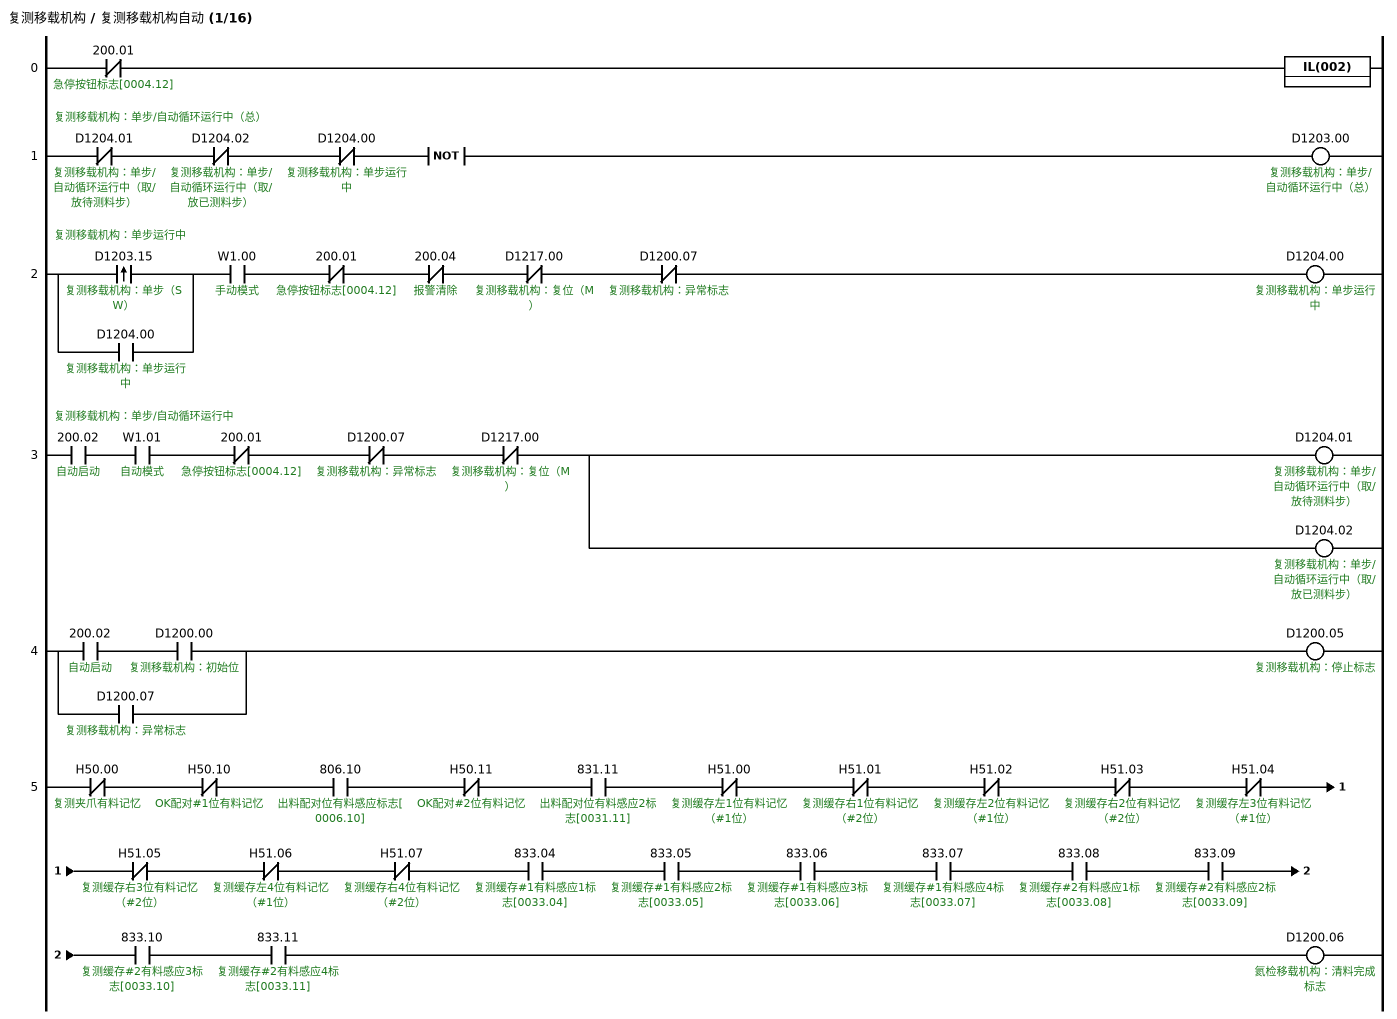
; [picture p528: 复测移载机构 / 复测移载机构自动, rungs 0-5]
; rung 0
LDNOT 200.01  ; 急停按钮标志[0004.12]
IL(002)
; rung 1: 复测移载机构：单步/自动循环运行中（总）
LDNOT D1204.01  ; 复测移载机构：单步/自动循环运行中（取/放待测料步）
ANDNOT D1204.02  ; 复测移载机构：单步/自动循环运行中（取/放已测料步）
ANDNOT D1204.00  ; 复测移载机构：单步运行中
NOT(520)
OUT D1203.00  ; 复测移载机构：单步/自动循环运行中（总）
; rung 2: 复测移载机构：单步运行中
@LD D1203.15  ; 复测移载机构：单步（SW）
OR D1204.00  ; 复测移载机构：单步运行中
AND W1.00  ; 手动模式
ANDNOT 200.01  ; 急停按钮标志[0004.12]
ANDNOT 200.04  ; 报警清除
ANDNOT D1217.00  ; 复测移载机构：复位（M）
ANDNOT D1200.07  ; 复测移载机构：异常标志
OUT D1204.00  ; 复测移载机构：单步运行中
; rung 3: 复测移载机构：单步/自动循环运行中
LD 200.02  ; 自动启动
AND W1.01  ; 自动模式
ANDNOT 200.01  ; 急停按钮标志[0004.12]
ANDNOT D1200.07  ; 复测移载机构：异常标志
ANDNOT D1217.00  ; 复测移载机构：复位（M）
OUT D1204.01  ; 复测移载机构：单步/自动循环运行中（取/放待测料步）
OUT D1204.02  ; 复测移载机构：单步/自动循环运行中（取/放已测料步）
; rung 4
LD 200.02  ; 自动启动
AND D1200.00  ; 复测移载机构：初始位
OR D1200.07  ; 复测移载机构：异常标志
OUT D1200.05  ; 复测移载机构：停止标志
; rung 5
LDNOT H50.00  ; 复测夹爪有料记忆
ANDNOT H50.10  ; OK配对#1位有料记忆
AND 806.10  ; 出料配对位有料感应标志[0006.10]
ANDNOT H50.11  ; OK配对#2位有料记忆
AND 831.11  ; 出料配对位有料感应2标志[0031.11]
ANDNOT H51.00  ; 复测缓存左1位有料记忆（#1位）
ANDNOT H51.01  ; 复测缓存右1位有料记忆（#2位）
ANDNOT H51.02  ; 复测缓存左2位有料记忆（#1位）
ANDNOT H51.03  ; 复测缓存右2位有料记忆（#2位）
ANDNOT H51.04  ; 复测缓存左3位有料记忆（#1位）
ANDNOT H51.05  ; 复测缓存右3位有料记忆（#2位）
ANDNOT H51.06  ; 复测缓存左4位有料记忆（#1位）
ANDNOT H51.07  ; 复测缓存右4位有料记忆（#2位）
AND 833.04  ; 复测缓存#1有料感应1标志[0033.04]
AND 833.05  ; 复测缓存#1有料感应2标志[0033.05]
AND 833.06  ; 复测缓存#1有料感应3标志[0033.06]
AND 833.07  ; 复测缓存#1有料感应4标志[0033.07]
AND 833.08  ; 复测缓存#2有料感应1标志[0033.08]
AND 833.09  ; 复测缓存#2有料感应2标志[0033.09]
AND 833.10  ; 复测缓存#2有料感应3标志[0033.10]
AND 833.11  ; 复测缓存#2有料感应4标志[0033.11]
OUT D1200.06  ; 氦检移载机构：清料完成标志

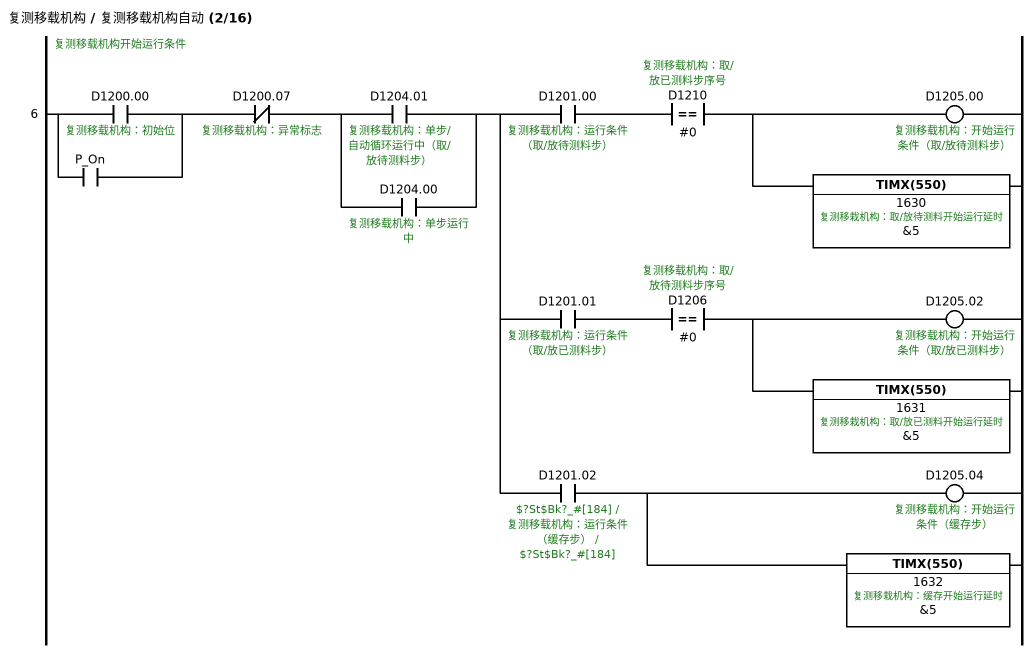
; rung 6: 复测移载机构开始运行条件
LD D1200.00  ; 复测移载机构：初始位
OR P_On
ANDNOT D1200.07  ; 复测移载机构：异常标志
LD D1204.01  ; 复测移载机构：单步/自动循环运行中（取/放待测料步）
OR D1204.00  ; 复测移载机构：单步运行中
ANDLD
OUT TR0
AND D1201.00  ; 复测移载机构：运行条件（取/放待测料步）
AND=L(301) D1210 #0  ; 复测移载机构：取/放已测料步序号
OUT D1205.00  ; 复测移载机构：开始运行条件（取/放待测料步）
TIMX(550) 1630 &5  ; 复测移栽机构：取/放待测料开始运行延时
LD TR0
AND D1201.01  ; 复测移载机构：运行条件（取/放已测料步）
AND=L(301) D1206 #0  ; 复测移载机构：取/放待测料步序号
OUT D1205.02  ; 复测移载机构：开始运行条件（取/放已测料步）
TIMX(550) 1631 &5  ; 复测移栽机构：取/放已测料开始运行延时
LD TR0
AND D1201.02  ; $?St$Bk?_#[184] / 复测移载机构：运行条件（缓存步） / $?St$Bk?_#[184]
OUT D1205.04  ; 复测移载机构：开始运行条件（缓存步）
TIMX(550) 1632 &5  ; 复测移栽机构：缓存开始运行延时

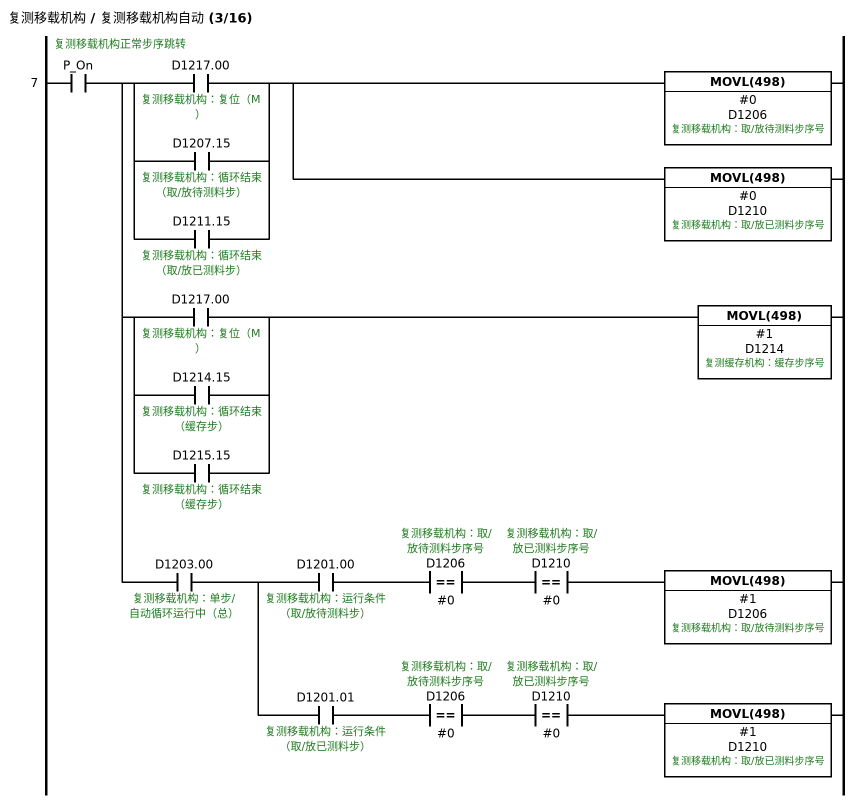
; rung 7: 复测移载机构正常步序跳转
LD P_On
OUT TR0
LD D1217.00  ; 复测移载机构：复位（M）
OR D1207.15  ; 复测移载机构：循环结束（取/放待测料步）
OR D1211.15  ; 复测移载机构：循环结束（取/放已测料步）
ANDLD
MOVL(498) #0 D1206  ; 复测移载机构：取/放待测料步序号
MOVL(498) #0 D1210  ; 复测移载机构：取/放已测料步序号
LD TR0
LD D1217.00  ; 复测移载机构：复位（M）
OR D1214.15  ; 复测移载机构：循环结束（缓存步）
OR D1215.15  ; 复测移载机构：循环结束（缓存步）
ANDLD
MOVL(498) #1 D1214  ; 复测缓存机构：缓存步序号
LD TR0
AND D1203.00  ; 复测移载机构：单步/自动循环运行中（总）
OUT TR0
AND D1201.00  ; 复测移载机构：运行条件（取/放待测料步）
AND=L(301) D1206 #0  ; 复测移载机构：取/放待测料步序号
AND=L(301) D1210 #0  ; 复测移载机构：取/放已测料步序号
MOVL(498) #1 D1206  ; 复测移载机构：取/放待测料步序号
LD TR0
AND D1201.01  ; 复测移载机构：运行条件（取/放已测料步）
AND=L(301) D1206 #0  ; 复测移载机构：取/放待测料步序号
AND=L(301) D1210 #0  ; 复测移载机构：取/放已测料步序号
MOVL(498) #1 D1210  ; 复测移载机构：取/放已测料步序号

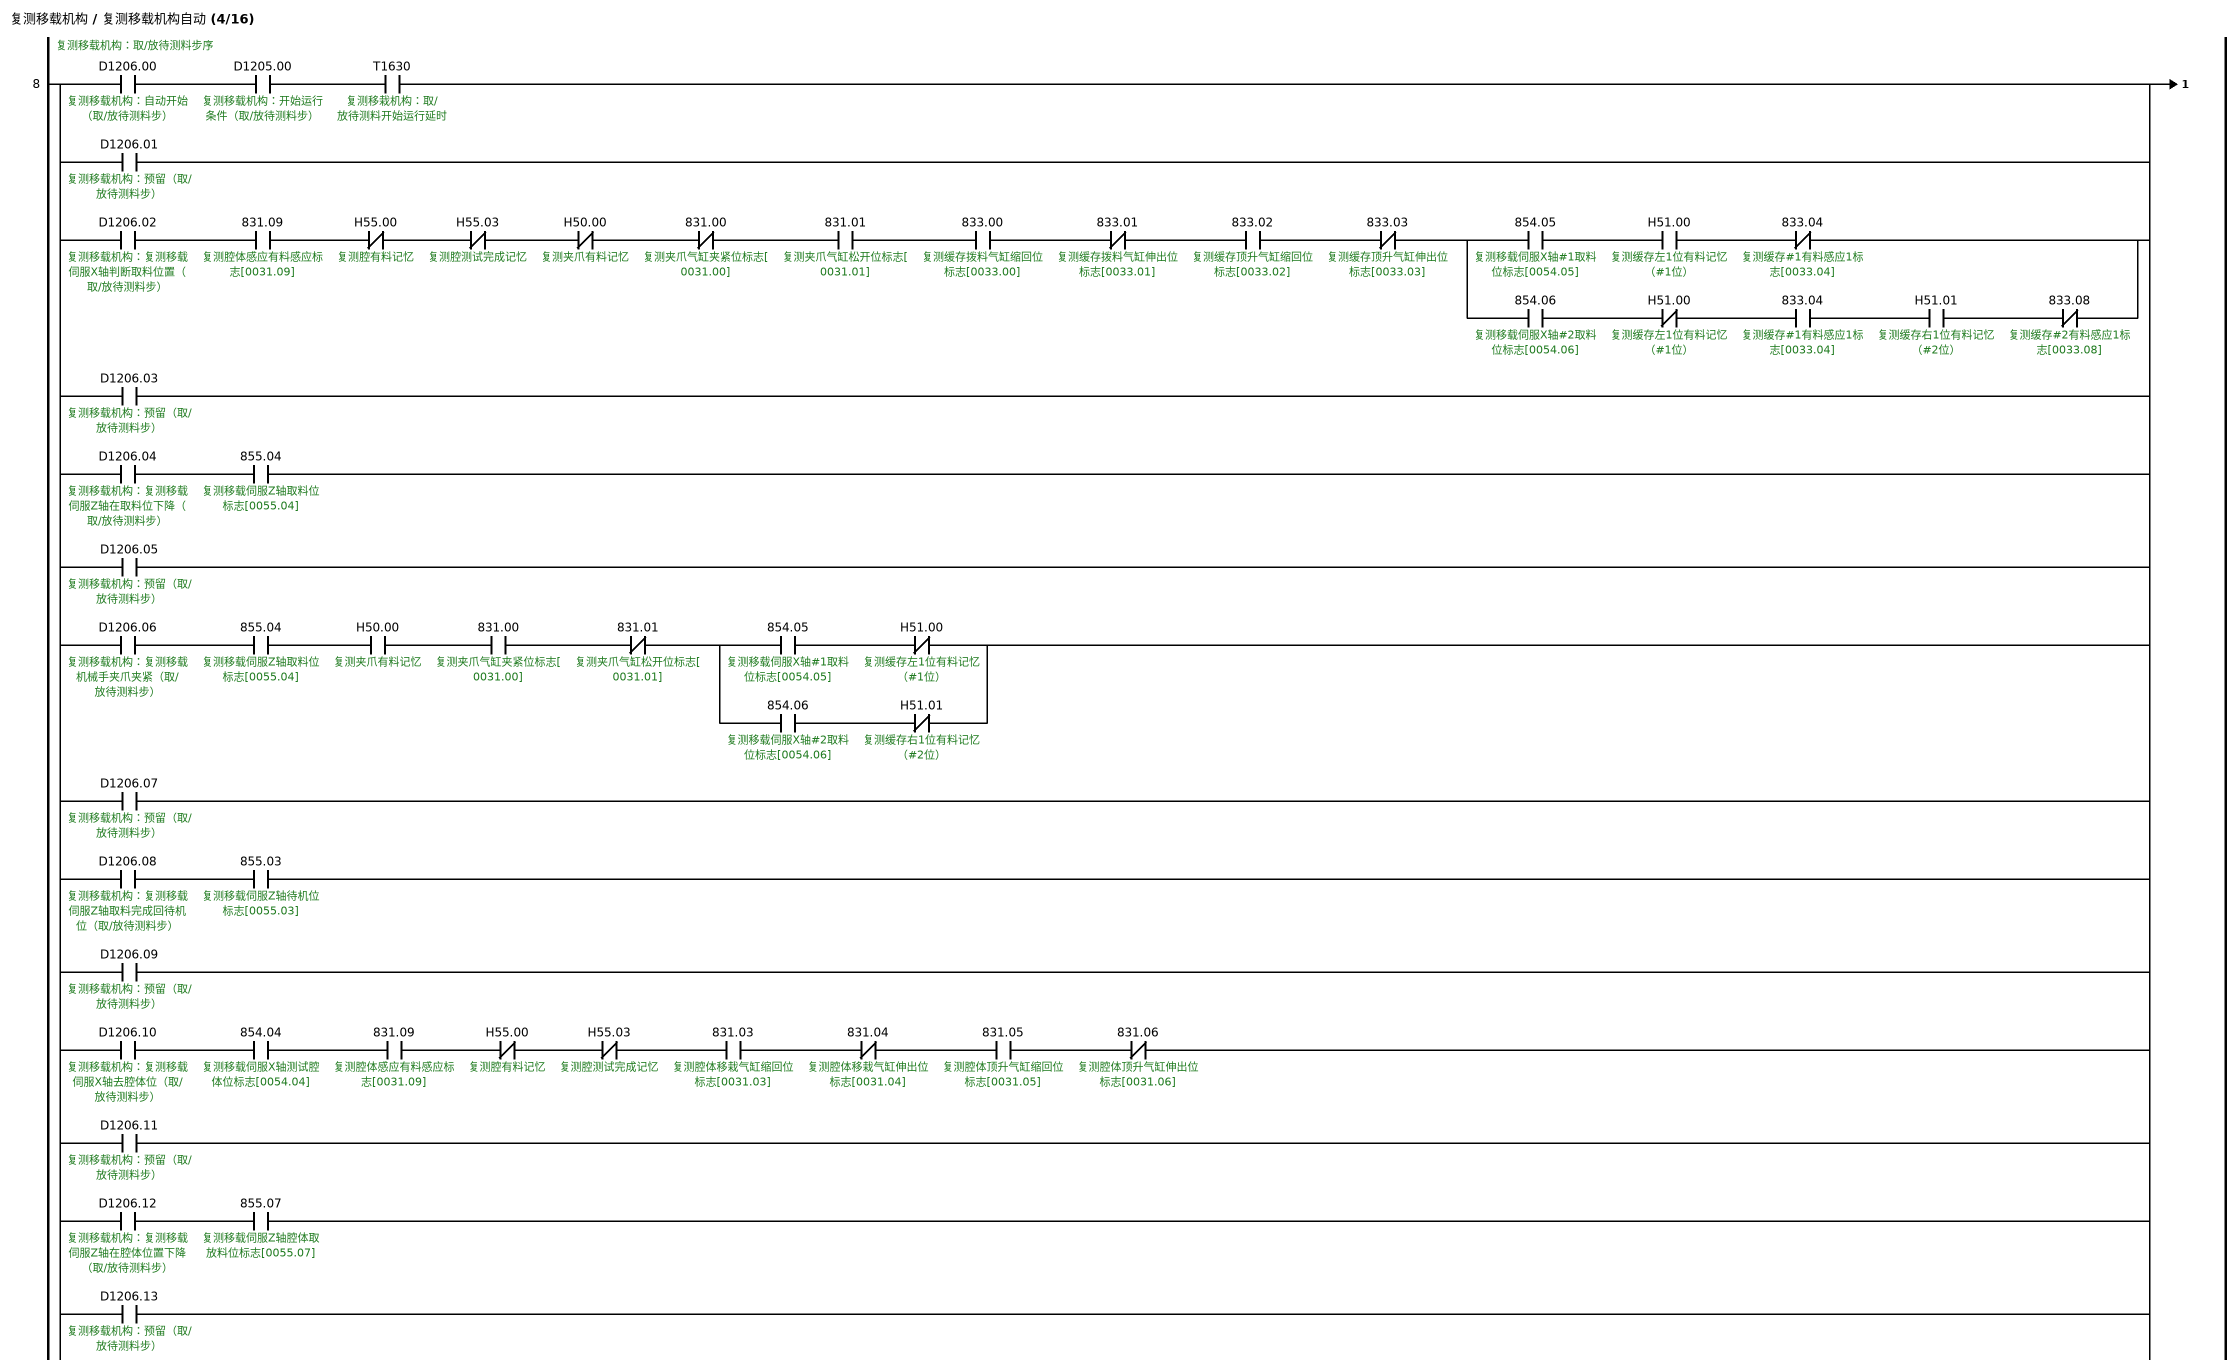

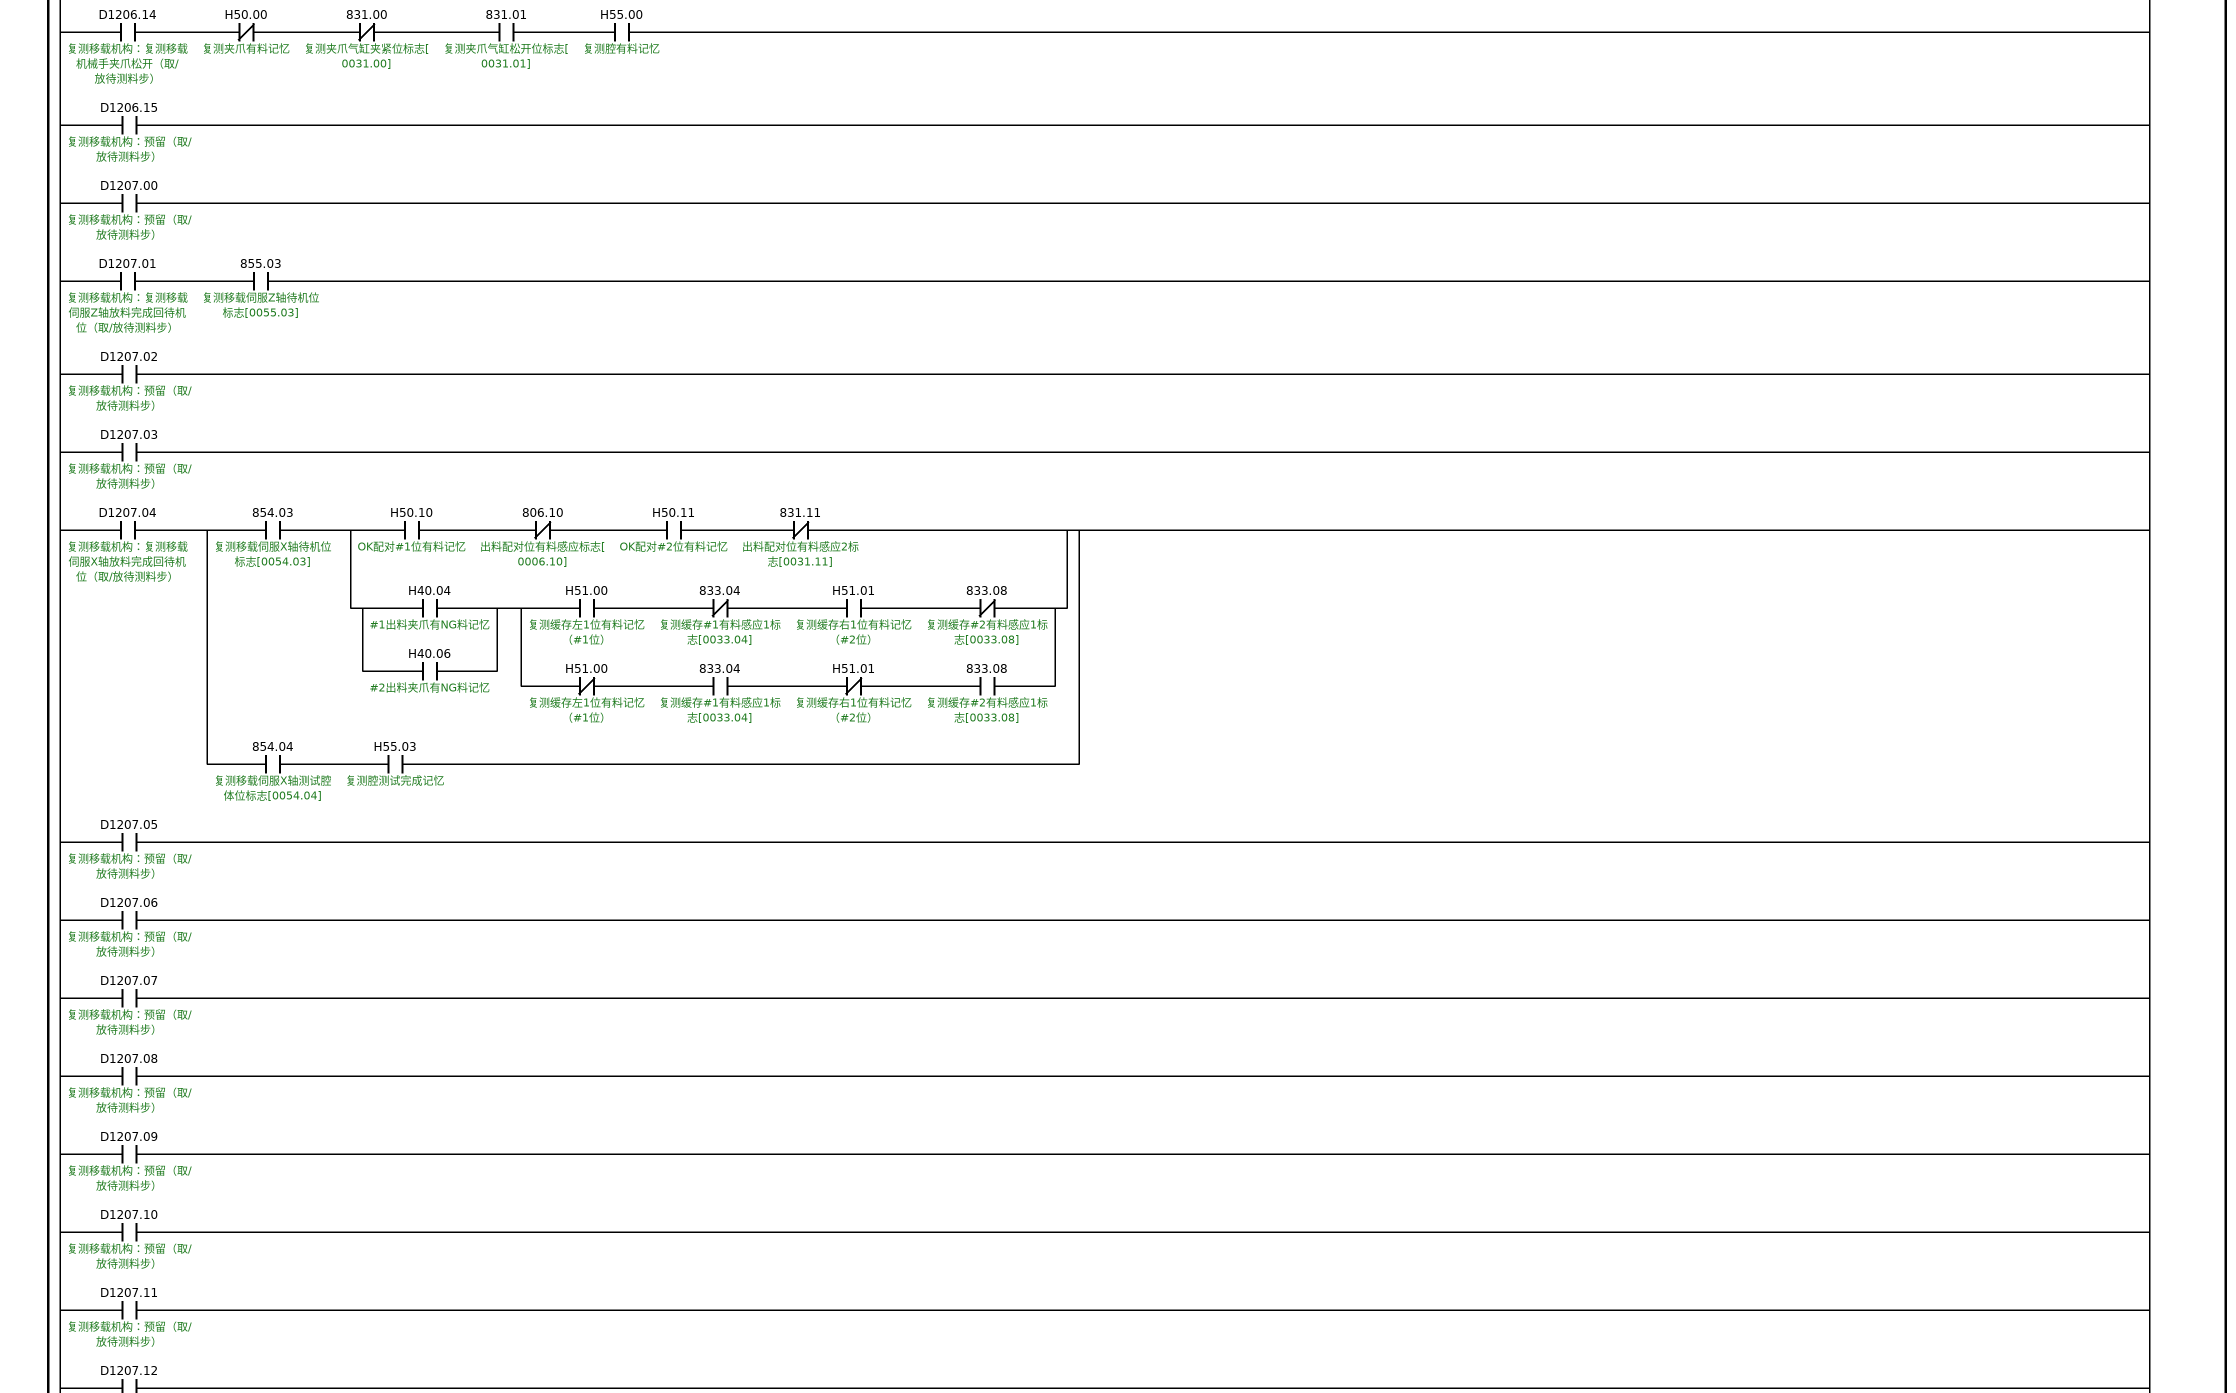

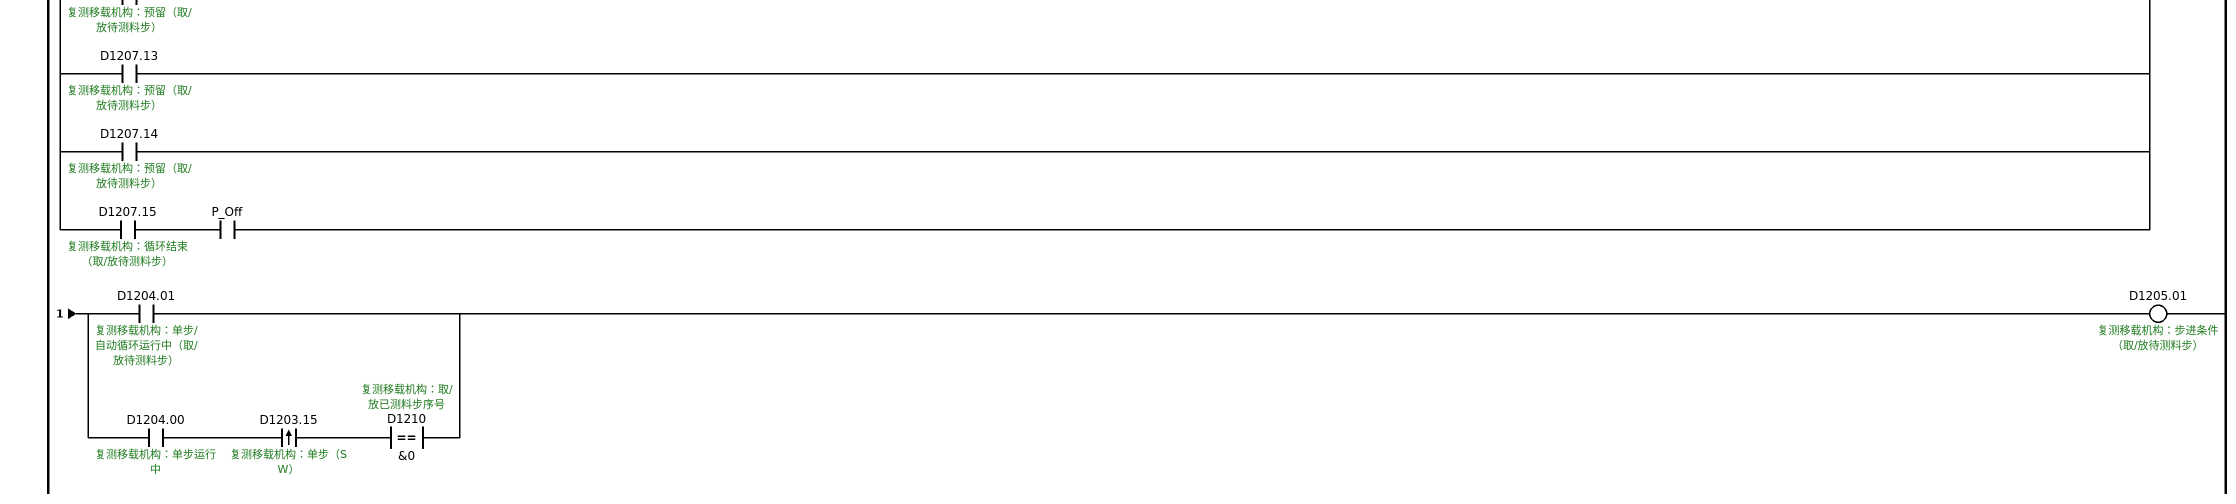
; rung 8: 复测移载机构：取/放待测料步序
LD D1206.00  ; 复测移载机构：自动开始（取/放待测料步）
AND D1205.00  ; 复测移载机构：开始运行条件（取/放待测料步）
AND T1630  ; 复测移栽机构：取/放待测料开始运行延时
OR D1206.01  ; 复测移载机构：预留（取/放待测料步）
LD D1206.02  ; 复测移载机构：复测移载伺服X轴判断取料位置（取/放待测料步）  // 如果出现带料初始化时，夹爪有料，则直接跳转至腔体放料步（D1206.10）
AND 831.09  ; 复测腔体感应有料感应标志[0031.09]
ANDNOT H55.00  ; 复测腔有料记忆
ANDNOT H55.03  ; 复测腔测试完成记忆
ANDNOT H50.00  ; 复测夹爪有料记忆
ANDNOT 831.00  ; 复测夹爪气缸夹紧位标志[0031.00]
AND 831.01  ; 复测夹爪气缸松开位标志[0031.01]
AND 833.00  ; 复测缓存拨料气缸缩回位标志[0033.00]
ANDNOT 833.01  ; 复测缓存拨料气缸伸出位标志[0033.01]
AND 833.02  ; 复测缓存顶升气缸缩回位标志[0033.02]
ANDNOT 833.03  ; 复测缓存顶升气缸伸出位标志[0033.03]
LD 854.05  ; 复测移载伺服X轴#1取料位标志[0054.05]
AND H51.00  ; 复测缓存左1位有料记忆（#1位）
ANDNOT 833.04  ; 复测缓存#1有料感应1标志[0033.04]
LD 854.06  ; 复测移载伺服X轴#2取料位标志[0054.06]
ANDNOT H51.00  ; 复测缓存左1位有料记忆（#1位）
AND 833.04  ; 复测缓存#1有料感应1标志[0033.04]
AND H51.01  ; 复测缓存右1位有料记忆（#2位）
ANDNOT 833.08  ; 复测缓存#2有料感应1标志[0033.08]
ORLD
ANDLD
ORLD
OR D1206.03  ; 复测移载机构：预留（取/放待测料步）
LD D1206.04  ; 复测移载机构：复测移载伺服Z轴在取料位下降（取/放待测料步）
AND 855.04  ; 复测移载伺服Z轴取料位标志[0055.04]
ORLD
OR D1206.05  ; 复测移载机构：预留（取/放待测料步）
LD D1206.06  ; 复测移载机构：复测移载机械手夹爪夹紧（取/放待测料步）
AND 855.04  ; 复测移载伺服Z轴取料位标志[0055.04]
AND H50.00  ; 复测夹爪有料记忆
AND 831.00  ; 复测夹爪气缸夹紧位标志[0031.00]
ANDNOT 831.01  ; 复测夹爪气缸松开位标志[0031.01]
LD 854.05  ; 复测移载伺服X轴#1取料位标志[0054.05]
ANDNOT H51.00  ; 复测缓存左1位有料记忆（#1位）
LD 854.06  ; 复测移载伺服X轴#2取料位标志[0054.06]
ANDNOT H51.01  ; 复测缓存右1位有料记忆（#2位）
ORLD
ANDLD
ORLD
OR D1206.07  ; 复测移载机构：预留（取/放待测料步）
LD D1206.08  ; 复测移载机构：复测移载伺服Z轴取料完成回待机位（取/放待测料步）
AND 855.03  ; 复测移载伺服Z轴待机位标志[0055.03]
ORLD
OR D1206.09  ; 复测移载机构：预留（取/放待测料步）
LD D1206.10  ; 复测移载机构：复测移载伺服X轴去腔体位（取/放待测料步）
AND 854.04  ; 复测移载伺服X轴测试腔体位标志[0054.04]
AND 831.09  ; 复测腔体感应有料感应标志[0031.09]
ANDNOT H55.00  ; 复测腔有料记忆
ANDNOT H55.03  ; 复测腔测试完成记忆
AND 831.03  ; 复测腔体移栽气缸缩回位标志[0031.03]
ANDNOT 831.04  ; 复测腔体移栽气缸伸出位标志[0031.04]
AND 831.05  ; 复测腔体顶升气缸缩回位标志[0031.05]
ANDNOT 831.06  ; 复测腔体顶升气缸伸出位标志[0031.06]
ORLD
OR D1206.11  ; 复测移载机构：预留（取/放待测料步）
LD D1206.12  ; 复测移载机构：复测移载伺服Z轴在腔体位置下降（取/放待测料步）
AND 855.07  ; 复测移载伺服Z轴腔体取放料位标志[0055.07]
ORLD
OR D1206.13  ; 复测移载机构：预留（取/放待测料步）
LD D1206.14  ; 复测移载机构：复测移载机械手夹爪松开（取/放待测料步）
ANDNOT H50.00  ; 复测夹爪有料记忆
ANDNOT 831.00  ; 复测夹爪气缸夹紧位标志[0031.00]
AND 831.01  ; 复测夹爪气缸松开位标志[0031.01]
AND H55.00  ; 复测腔有料记忆
ORLD
OR D1206.15  ; 复测移载机构：预留（取/放待测料步）
OR D1207.00  ; 复测移载机构：预留（取/放待测料步）
LD D1207.01  ; 复测移载机构：复测移载伺服Z轴放料完成回待机位（取/放待测料步）
AND 855.03  ; 复测移载伺服Z轴待机位标志[0055.03]
ORLD
OR D1207.02  ; 复测移载机构：预留（取/放待测料步）
OR D1207.03  ; 复测移载机构：预留（取/放待测料步）
LD D1207.04  ; 复测移载机构：复测移载伺服X轴放料完成回待机位（取/放待测料步）  // 当配对位有空位，且缓存位有单料时在腔体位等待
LD 854.03  ; 复测移载伺服X轴待机位标志[0054.03]
LD H50.10  ; OK配对#1位有料记忆
ANDNOT 806.10  ; 出料配对位有料感应标志[0006.10]
AND H50.11  ; OK配对#2位有料记忆
ANDNOT 831.11  ; 出料配对位有料感应2标志[0031.11]
LD H40.04  ; #1出料夹爪有NG料记忆
OR H40.06  ; #2出料夹爪有NG料记忆
LD H51.00  ; 复测缓存左1位有料记忆（#1位）
ANDNOT 833.04  ; 复测缓存#1有料感应1标志[0033.04]
AND H51.01  ; 复测缓存右1位有料记忆（#2位）
ANDNOT 833.08  ; 复测缓存#2有料感应1标志[0033.08]
LDNOT H51.00  ; 复测缓存左1位有料记忆（#1位）
AND 833.04  ; 复测缓存#1有料感应1标志[0033.04]
ANDNOT H51.01  ; 复测缓存右1位有料记忆（#2位）
AND 833.08  ; 复测缓存#2有料感应1标志[0033.08]
ORLD
ANDLD
ORLD
ANDLD
LD 854.04  ; 复测移载伺服X轴测试腔体位标志[0054.04]
AND H55.03  ; 复测腔测试完成记忆
ORLD
ANDLD
ORLD
OR D1207.05  ; 复测移载机构：预留（取/放待测料步）
OR D1207.06  ; 复测移载机构：预留（取/放待测料步）
OR D1207.07  ; 复测移载机构：预留（取/放待测料步）
OR D1207.08  ; 复测移载机构：预留（取/放待测料步）
OR D1207.09  ; 复测移载机构：预留（取/放待测料步）
OR D1207.10  ; 复测移载机构：预留（取/放待测料步）
OR D1207.11  ; 复测移载机构：预留（取/放待测料步）
OR D1207.12  ; 复测移载机构：预留（取/放待测料步）
OR D1207.13  ; 复测移载机构：预留（取/放待测料步）
OR D1207.14  ; 复测移载机构：预留（取/放待测料步）
LD D1207.15  ; 复测移载机构：循环结束（取/放待测料步）
AND P_Off
ORLD
LD D1204.01  ; 复测移载机构：单步/自动循环运行中（取/放待测料步）
LD D1204.00  ; 复测移载机构：单步运行中
@AND D1203.15  ; 复测移载机构：单步（SW）
AND=L(301) D1210 &0  ; 复测移载机构：取/放已测料步序号
ORLD
ANDLD
OUT D1205.01  ; 复测移载机构：步进条件（取/放待测料步）

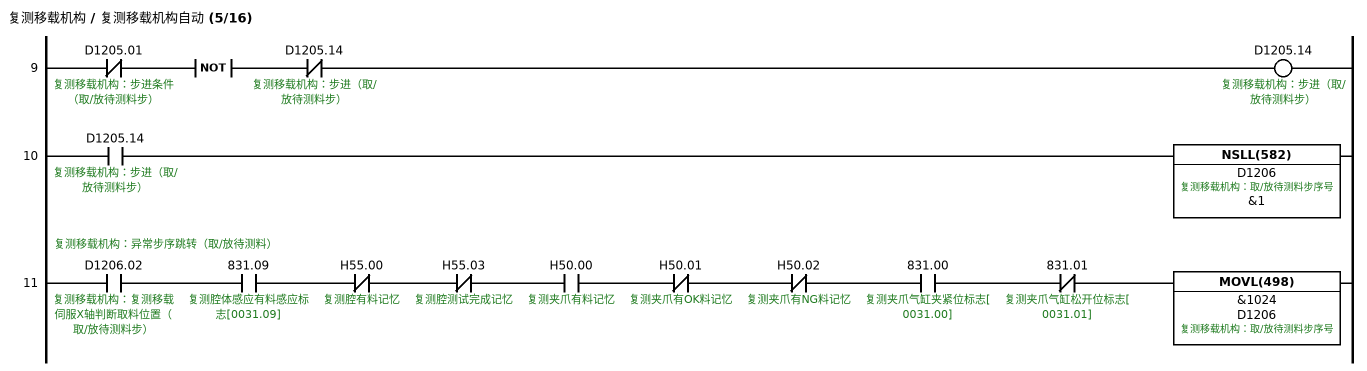
; rung 9
LDNOT D1205.01  ; 复测移载机构：步进条件（取/放待测料步）
NOT(520)
ANDNOT D1205.14  ; 复测移载机构：步进（取/放待测料步）
OUT D1205.14  ; 复测移载机构：步进（取/放待测料步）
; rung 10
LD D1205.14  ; 复测移载机构：步进（取/放待测料步）
NSLL(582) D1206 &1  ; 复测移载机构：取/放待测料步序号
; rung 11: 复测移载机构：异常步序跳转（取/放待测料）
LD D1206.02  ; 复测移载机构：复测移载伺服X轴判断取料位置（取/放待测料步）  // 如果出现带料初始化时，夹爪有料，则直接跳转至腔体放料步（D1206.10）
AND 831.09  ; 复测腔体感应有料感应标志[0031.09]
ANDNOT H55.00  ; 复测腔有料记忆
ANDNOT H55.03  ; 复测腔测试完成记忆
AND H50.00  ; 复测夹爪有料记忆
ANDNOT H50.01  ; 复测夹爪有OK料记忆
ANDNOT H50.02  ; 复测夹爪有NG料记忆
AND 831.00  ; 复测夹爪气缸夹紧位标志[0031.00]
ANDNOT 831.01  ; 复测夹爪气缸松开位标志[0031.01]
MOVL(498) &1024 D1206  ; 复测移载机构：取/放待测料步序号

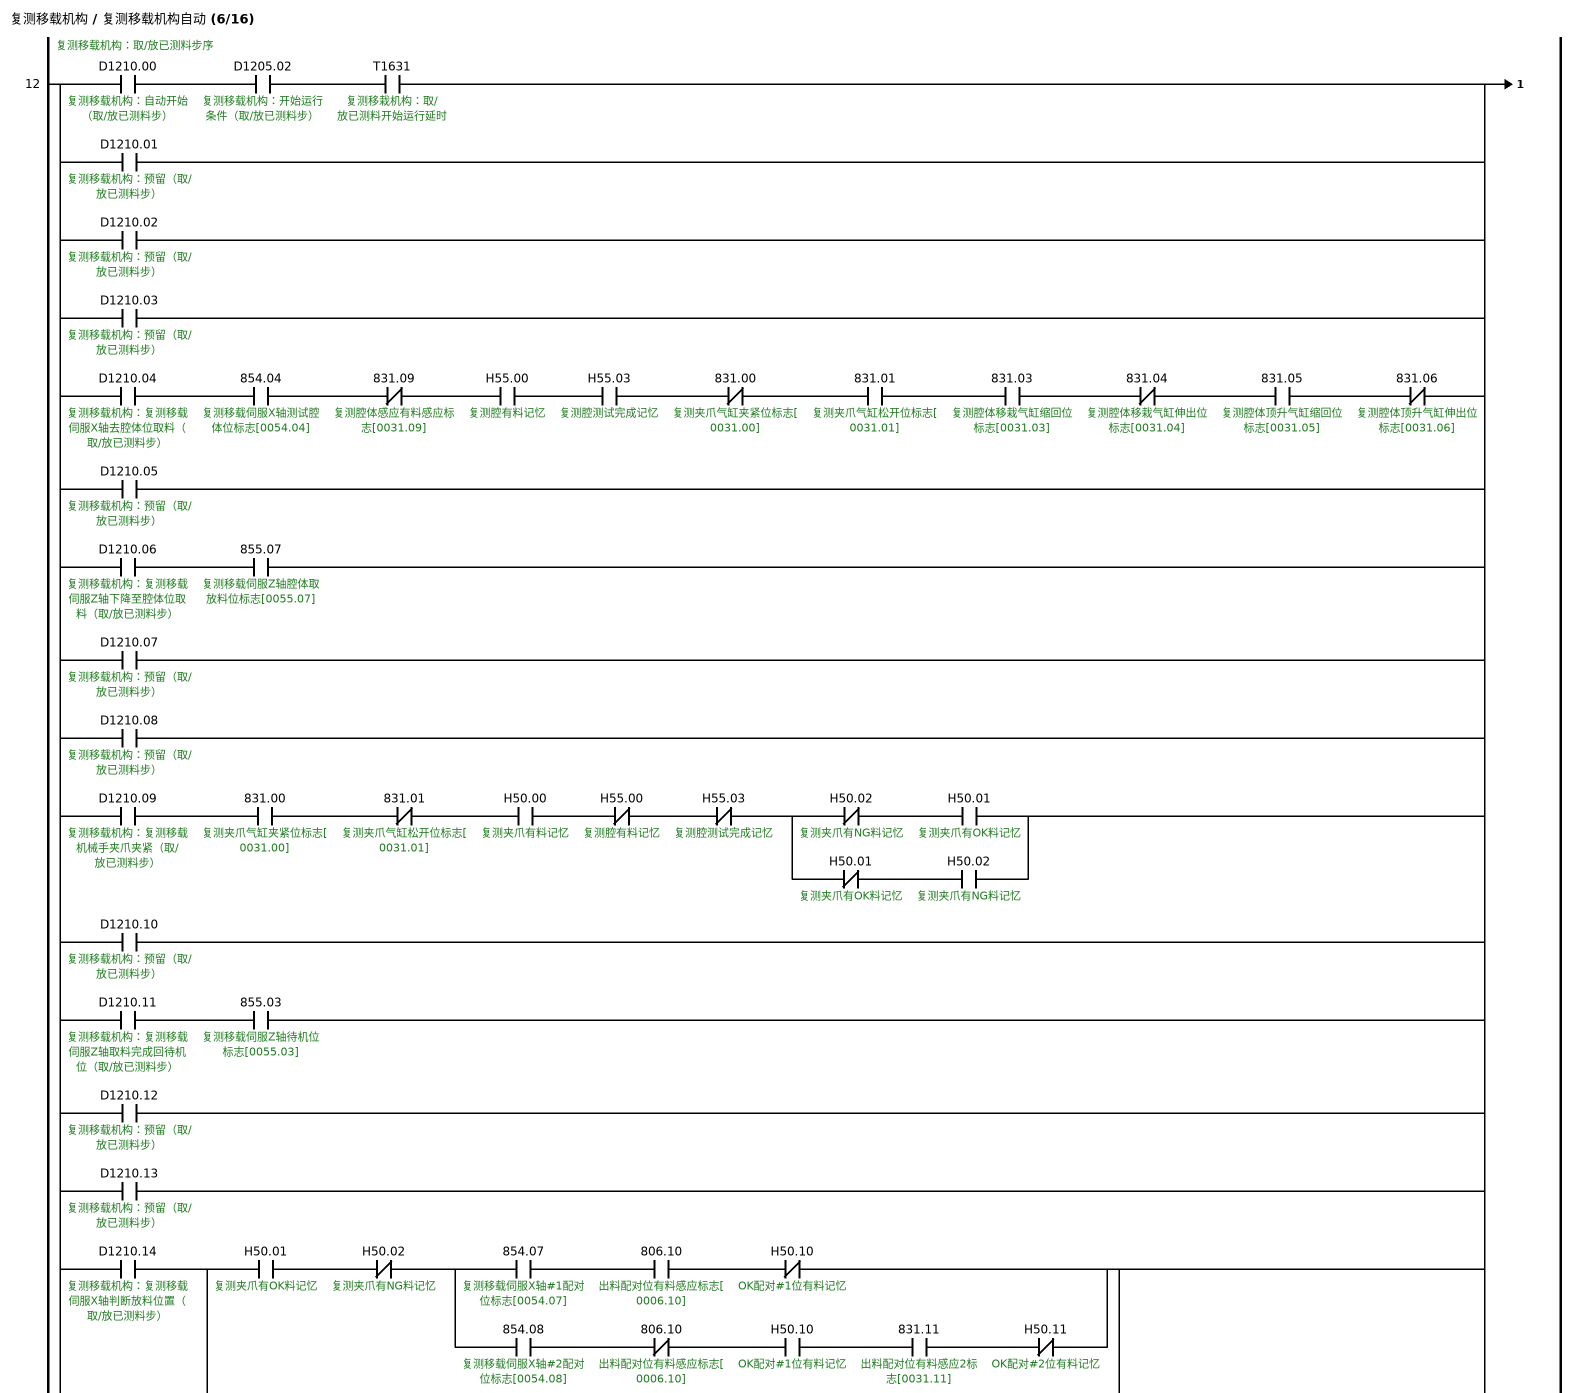

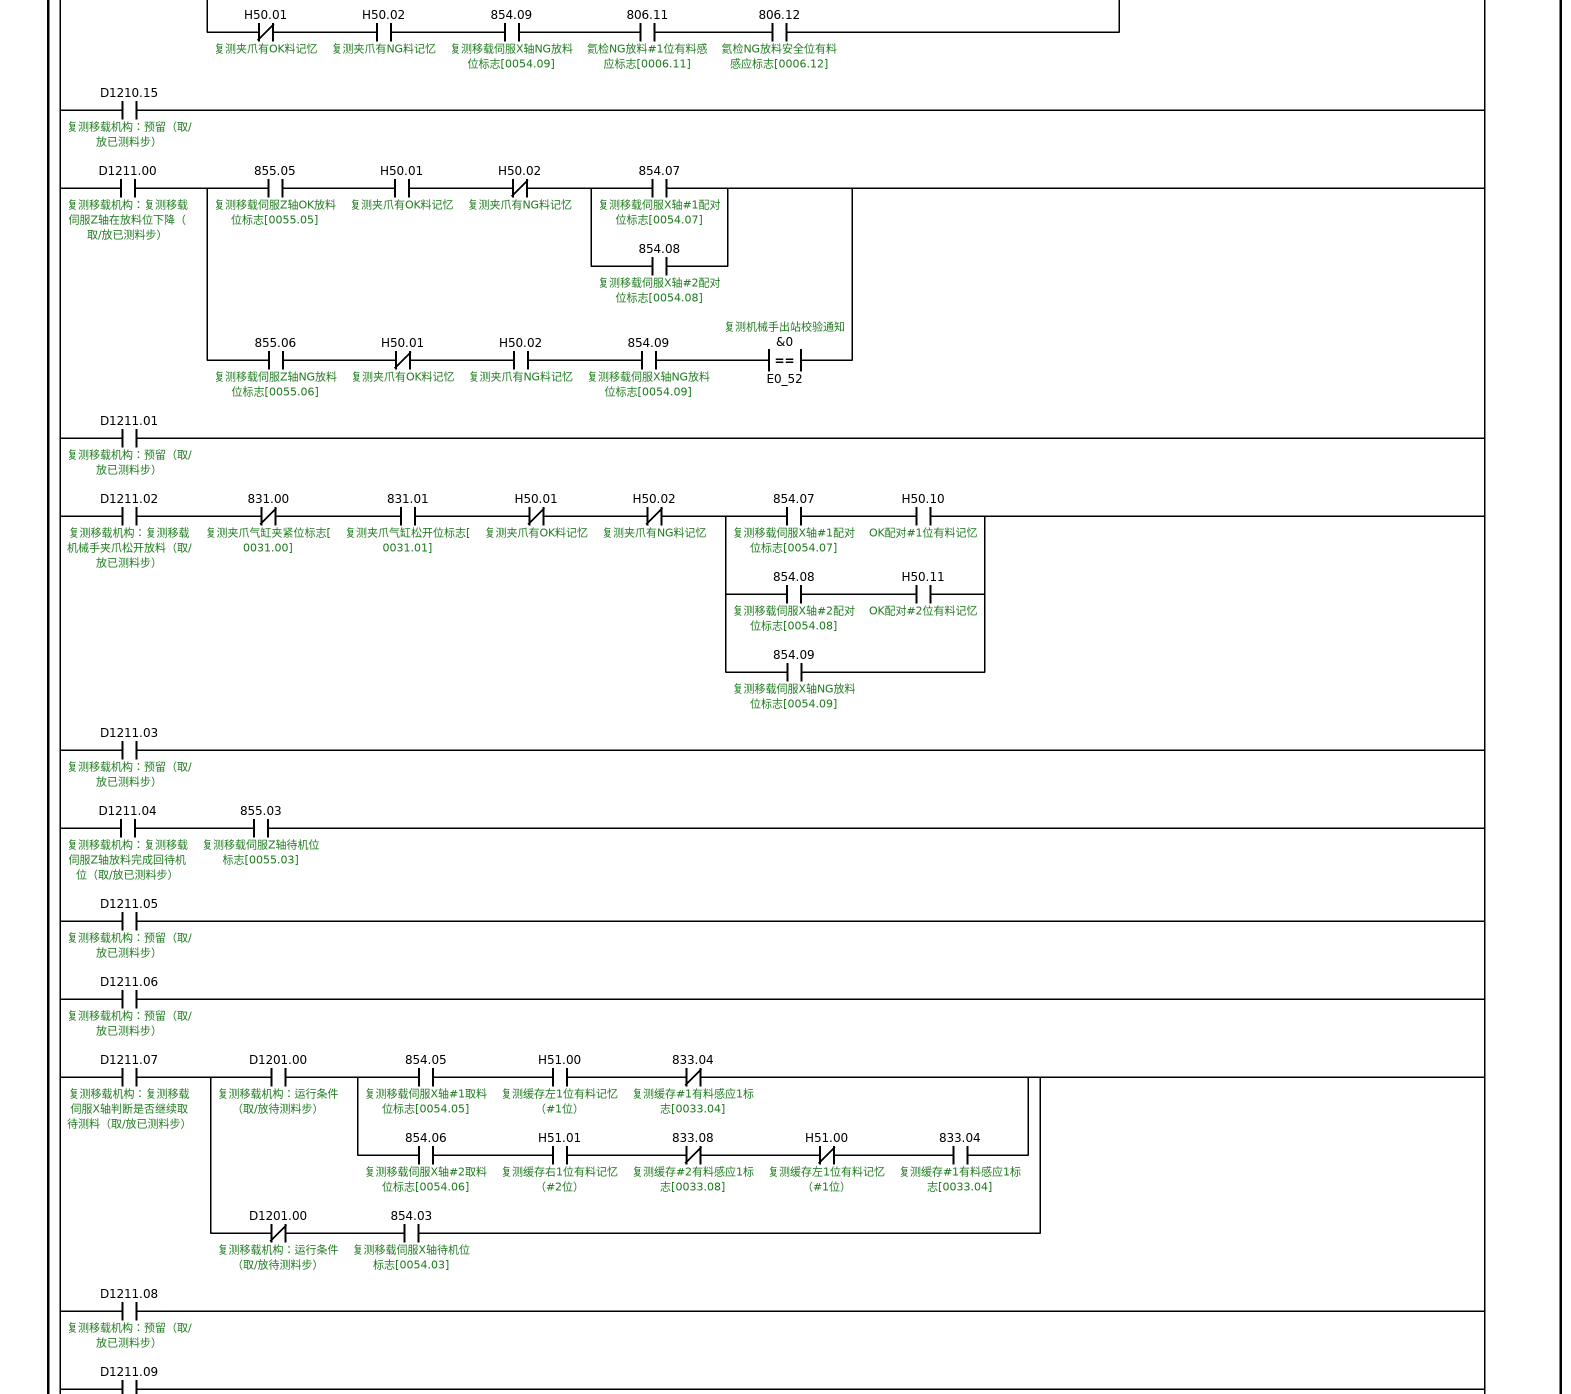

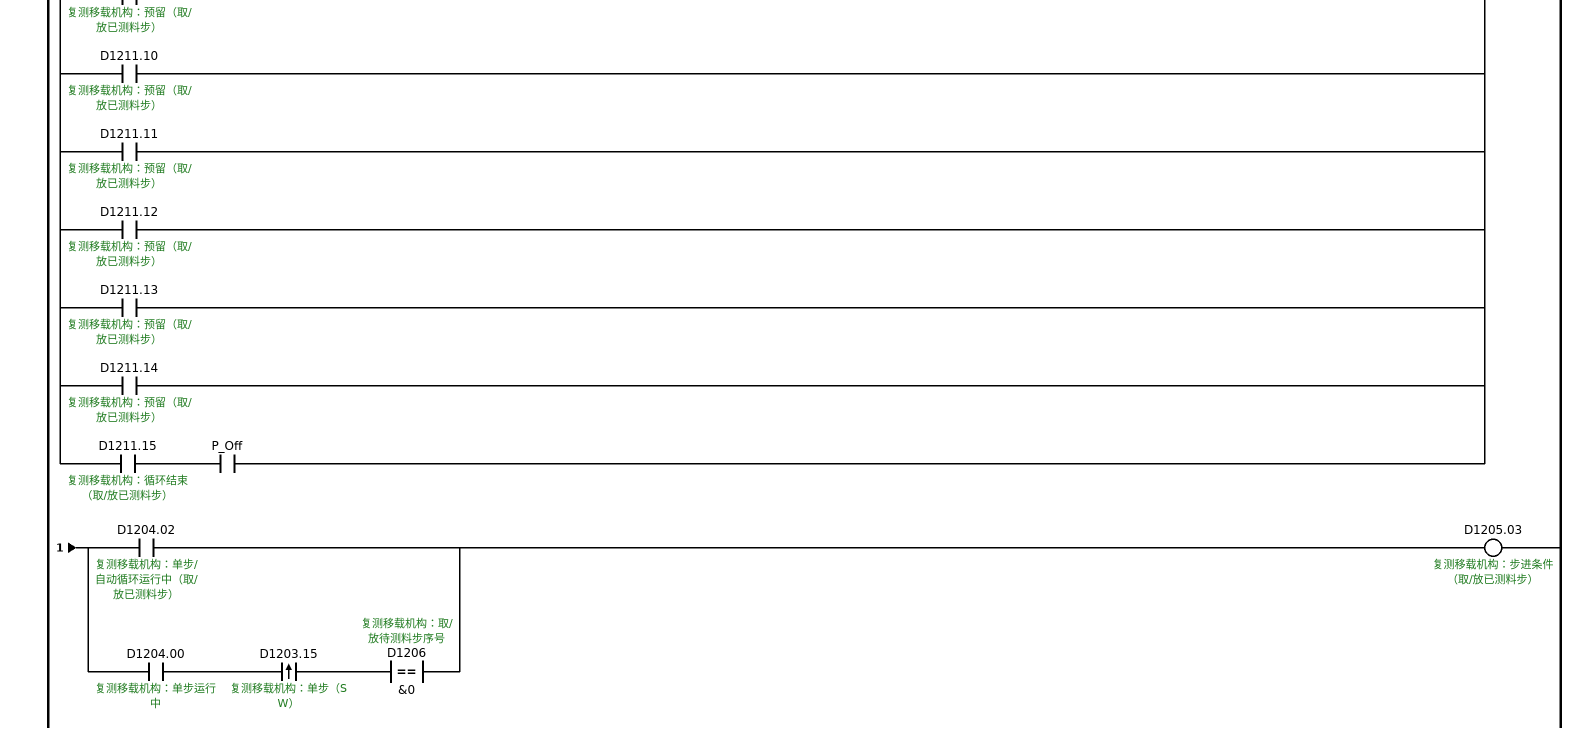
; rung 12: 复测移载机构：取/放已测料步序
LD D1210.00  ; 复测移载机构：自动开始（取/放已测料步）
AND D1205.02  ; 复测移载机构：开始运行条件（取/放已测料步）
AND T1631  ; 复测移栽机构：取/放已测料开始运行延时
OR D1210.01  ; 复测移载机构：预留（取/放已测料步）
OR D1210.02  ; 复测移载机构：预留（取/放已测料步）
OR D1210.03  ; 复测移载机构：预留（取/放已测料步）
LD D1210.04  ; 复测移载机构：复测移载伺服X轴去腔体位取料（取/放已测料步）  // 如果出现带料初始化时，夹爪有料，则直接跳转至放料判断步（D1210.14）
AND 854.04  ; 复测移载伺服X轴测试腔体位标志[0054.04]
ANDNOT 831.09  ; 复测腔体感应有料感应标志[0031.09]
AND H55.00  ; 复测腔有料记忆
AND H55.03  ; 复测腔测试完成记忆
ANDNOT 831.00  ; 复测夹爪气缸夹紧位标志[0031.00]
AND 831.01  ; 复测夹爪气缸松开位标志[0031.01]
AND 831.03  ; 复测腔体移栽气缸缩回位标志[0031.03]
ANDNOT 831.04  ; 复测腔体移栽气缸伸出位标志[0031.04]
AND 831.05  ; 复测腔体顶升气缸缩回位标志[0031.05]
ANDNOT 831.06  ; 复测腔体顶升气缸伸出位标志[0031.06]
ORLD
OR D1210.05  ; 复测移载机构：预留（取/放已测料步）
LD D1210.06  ; 复测移载机构：复测移载伺服Z轴下降至腔体位取料（取/放已测料步）
AND 855.07  ; 复测移载伺服Z轴腔体取放料位标志[0055.07]
ORLD
OR D1210.07  ; 复测移载机构：预留（取/放已测料步）
OR D1210.08  ; 复测移载机构：预留（取/放已测料步）
LD D1210.09  ; 复测移载机构：复测移载机械手夹爪夹紧（取/放已测料步）
AND 831.00  ; 复测夹爪气缸夹紧位标志[0031.00]
ANDNOT 831.01  ; 复测夹爪气缸松开位标志[0031.01]
AND H50.00  ; 复测夹爪有料记忆
ANDNOT H55.00  ; 复测腔有料记忆
ANDNOT H55.03  ; 复测腔测试完成记忆
LDNOT H50.02  ; 复测夹爪有NG料记忆
AND H50.01  ; 复测夹爪有OK料记忆
LDNOT H50.01  ; 复测夹爪有OK料记忆
AND H50.02  ; 复测夹爪有NG料记忆
ORLD
ANDLD
ORLD
OR D1210.10  ; 复测移载机构：预留（取/放已测料步）
LD D1210.11  ; 复测移载机构：复测移载伺服Z轴取料完成回待机位（取/放已测料步）
AND 855.03  ; 复测移载伺服Z轴待机位标志[0055.03]
ORLD
OR D1210.12  ; 复测移载机构：预留（取/放已测料步）
OR D1210.13  ; 复测移载机构：预留（取/放已测料步）
LD D1210.14  ; 复测移载机构：复测移载伺服X轴判断放料位置（取/放已测料步）
LD H50.01  ; 复测夹爪有OK料记忆
ANDNOT H50.02  ; 复测夹爪有NG料记忆
LD 854.07  ; 复测移载伺服X轴#1配对位标志[0054.07]
AND 806.10  ; 出料配对位有料感应标志[0006.10]
ANDNOT H50.10  ; OK配对#1位有料记忆
LD 854.08  ; 复测移载伺服X轴#2配对位标志[0054.08]
ANDNOT 806.10  ; 出料配对位有料感应标志[0006.10]
AND H50.10  ; OK配对#1位有料记忆
AND 831.11  ; 出料配对位有料感应2标志[0031.11]
ANDNOT H50.11  ; OK配对#2位有料记忆
ORLD
ANDLD
LDNOT H50.01  ; 复测夹爪有OK料记忆
AND H50.02  ; 复测夹爪有NG料记忆
AND 854.09  ; 复测移载伺服X轴NG放料位标志[0054.09]
AND 806.11  ; 氦检NG放料#1位有料感应标志[0006.11]
AND 806.12  ; 氦检NG放料安全位有料感应标志[0006.12]
ORLD
ANDLD
ORLD
OR D1210.15  ; 复测移载机构：预留（取/放已测料步）
LD D1211.00  ; 复测移载机构：复测移载伺服Z轴在放料位下降（取/放已测料步）
LD 855.05  ; 复测移载伺服Z轴OK放料位标志[0055.05]
AND H50.01  ; 复测夹爪有OK料记忆
ANDNOT H50.02  ; 复测夹爪有NG料记忆
LD 854.07  ; 复测移载伺服X轴#1配对位标志[0054.07]
OR 854.08  ; 复测移载伺服X轴#2配对位标志[0054.08]
ANDLD
LD 855.06  ; 复测移载伺服Z轴NG放料位标志[0055.06]
ANDNOT H50.01  ; 复测夹爪有OK料记忆
AND H50.02  ; 复测夹爪有NG料记忆
AND 854.09  ; 复测移载伺服X轴NG放料位标志[0054.09]
AND=(300) &0 E0_52  ; 复测机械手出站校验通知
ORLD
ANDLD
ORLD
OR D1211.01  ; 复测移载机构：预留（取/放已测料步）
LD D1211.02  ; 复测移载机构：复测移载机械手夹爪松开放料（取/放已测料步）
ANDNOT 831.00  ; 复测夹爪气缸夹紧位标志[0031.00]
AND 831.01  ; 复测夹爪气缸松开位标志[0031.01]
ANDNOT H50.01  ; 复测夹爪有OK料记忆
ANDNOT H50.02  ; 复测夹爪有NG料记忆
LD 854.07  ; 复测移载伺服X轴#1配对位标志[0054.07]
AND H50.10  ; OK配对#1位有料记忆
LD 854.08  ; 复测移载伺服X轴#2配对位标志[0054.08]
AND H50.11  ; OK配对#2位有料记忆
ORLD
OR 854.09  ; 复测移载伺服X轴NG放料位标志[0054.09]
ANDLD
ORLD
OR D1211.03  ; 复测移载机构：预留（取/放已测料步）
LD D1211.04  ; 复测移载机构：复测移载伺服Z轴放料完成回待机位（取/放已测料步）
AND 855.03  ; 复测移载伺服Z轴待机位标志[0055.03]
ORLD
OR D1211.05  ; 复测移载机构：预留（取/放已测料步）
OR D1211.06  ; 复测移载机构：预留（取/放已测料步）
LD D1211.07  ; 复测移载机构：复测移载伺服X轴判断是否继续取待测料（取/放已测料步）  // 如还有待测料取料需求，则直接从放料位回到取料位，无待测料取料需求则直接回待机位
LD D1201.00  ; 复测移载机构：运行条件（取/放待测料步）
LD 854.05  ; 复测移载伺服X轴#1取料位标志[0054.05]
AND H51.00  ; 复测缓存左1位有料记忆（#1位）
ANDNOT 833.04  ; 复测缓存#1有料感应1标志[0033.04]
LD 854.06  ; 复测移载伺服X轴#2取料位标志[0054.06]
AND H51.01  ; 复测缓存右1位有料记忆（#2位）
ANDNOT 833.08  ; 复测缓存#2有料感应1标志[0033.08]
ANDNOT H51.00  ; 复测缓存左1位有料记忆（#1位）
AND 833.04  ; 复测缓存#1有料感应1标志[0033.04]
ORLD
ANDLD
LDNOT D1201.00  ; 复测移载机构：运行条件（取/放待测料步）
AND 854.03  ; 复测移载伺服X轴待机位标志[0054.03]
ORLD
ANDLD
ORLD
OR D1211.08  ; 复测移载机构：预留（取/放已测料步）
OR D1211.09  ; 复测移载机构：预留（取/放已测料步）
OR D1211.10  ; 复测移载机构：预留（取/放已测料步）
OR D1211.11  ; 复测移载机构：预留（取/放已测料步）
OR D1211.12  ; 复测移载机构：预留（取/放已测料步）
OR D1211.13  ; 复测移载机构：预留（取/放已测料步）
OR D1211.14  ; 复测移载机构：预留（取/放已测料步）
LD D1211.15  ; 复测移载机构：循环结束（取/放已测料步）
AND P_Off
ORLD
LD D1204.02  ; 复测移载机构：单步/自动循环运行中（取/放已测料步）
LD D1204.00  ; 复测移载机构：单步运行中
@AND D1203.15  ; 复测移载机构：单步（SW）
AND=L(301) D1206 &0  ; 复测移载机构：取/放待测料步序号
ORLD
ANDLD
OUT D1205.03  ; 复测移载机构：步进条件（取/放已测料步）

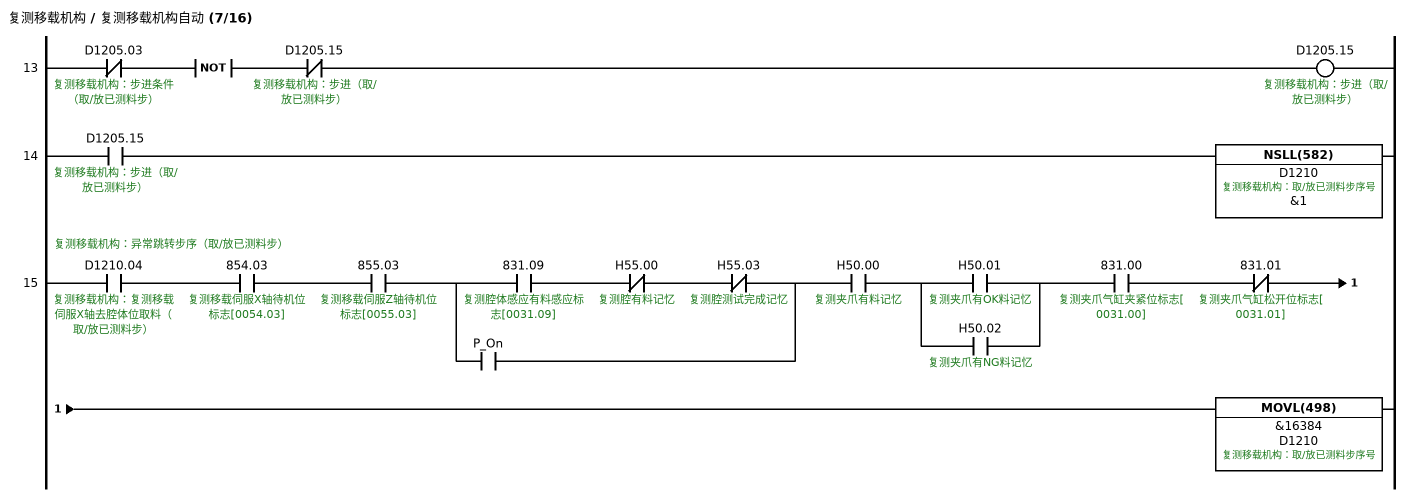
; rung 13
LDNOT D1205.03  ; 复测移载机构：步进条件（取/放已测料步）
NOT(520)
ANDNOT D1205.15  ; 复测移载机构：步进（取/放已测料步）
OUT D1205.15  ; 复测移载机构：步进（取/放已测料步）
; rung 14
LD D1205.15  ; 复测移载机构：步进（取/放已测料步）
NSLL(582) D1210 &1  ; 复测移载机构：取/放已测料步序号
; rung 15: 复测移载机构：异常跳转步序（取/放已测料步）
LD D1210.04  ; 复测移载机构：复测移载伺服X轴去腔体位取料（取/放已测料步）  // 如果出现带料初始化时，夹爪有料，则直接跳转至放料判断步（D1210.14）
AND 854.03  ; 复测移载伺服X轴待机位标志[0054.03]
AND 855.03  ; 复测移载伺服Z轴待机位标志[0055.03]
LD 831.09  ; 复测腔体感应有料感应标志[0031.09]
ANDNOT H55.00  ; 复测腔有料记忆
ANDNOT H55.03  ; 复测腔测试完成记忆
OR P_On
ANDLD
AND H50.00  ; 复测夹爪有料记忆
LD H50.01  ; 复测夹爪有OK料记忆
OR H50.02  ; 复测夹爪有NG料记忆
ANDLD
AND 831.00  ; 复测夹爪气缸夹紧位标志[0031.00]
ANDNOT 831.01  ; 复测夹爪气缸松开位标志[0031.01]
MOVL(498) &16384 D1210  ; 复测移载机构：取/放已测料步序号

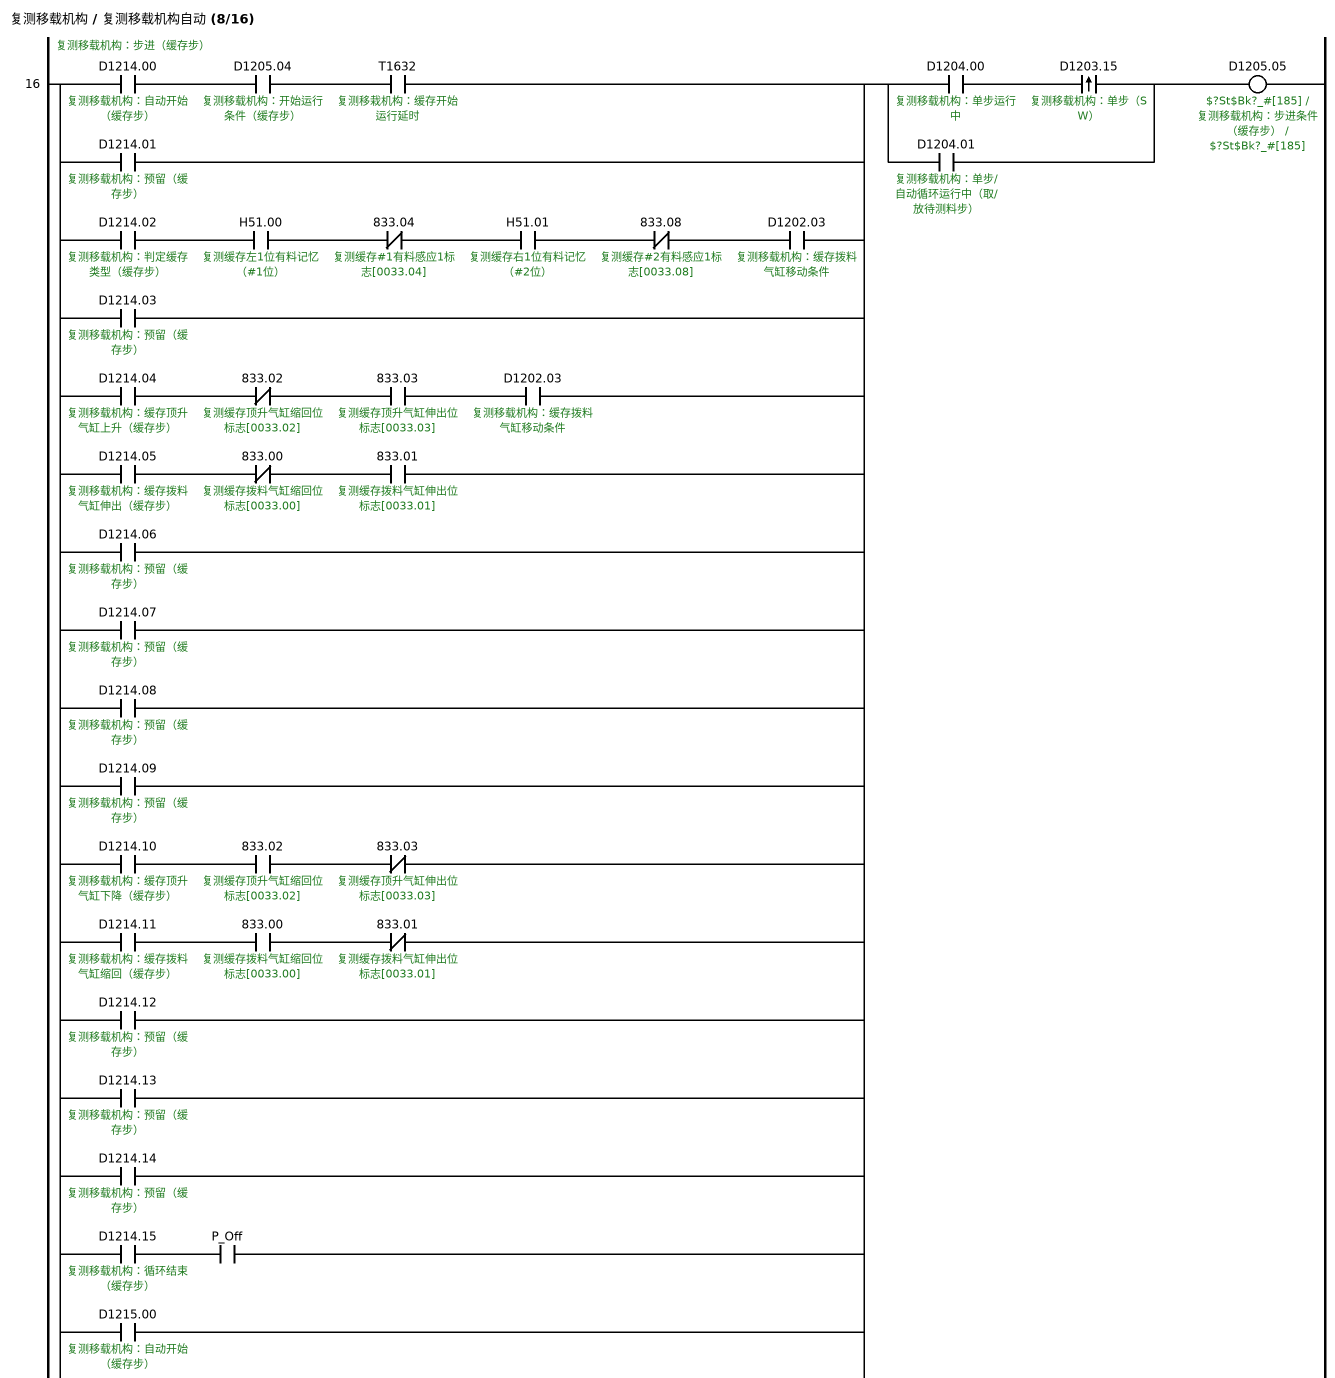

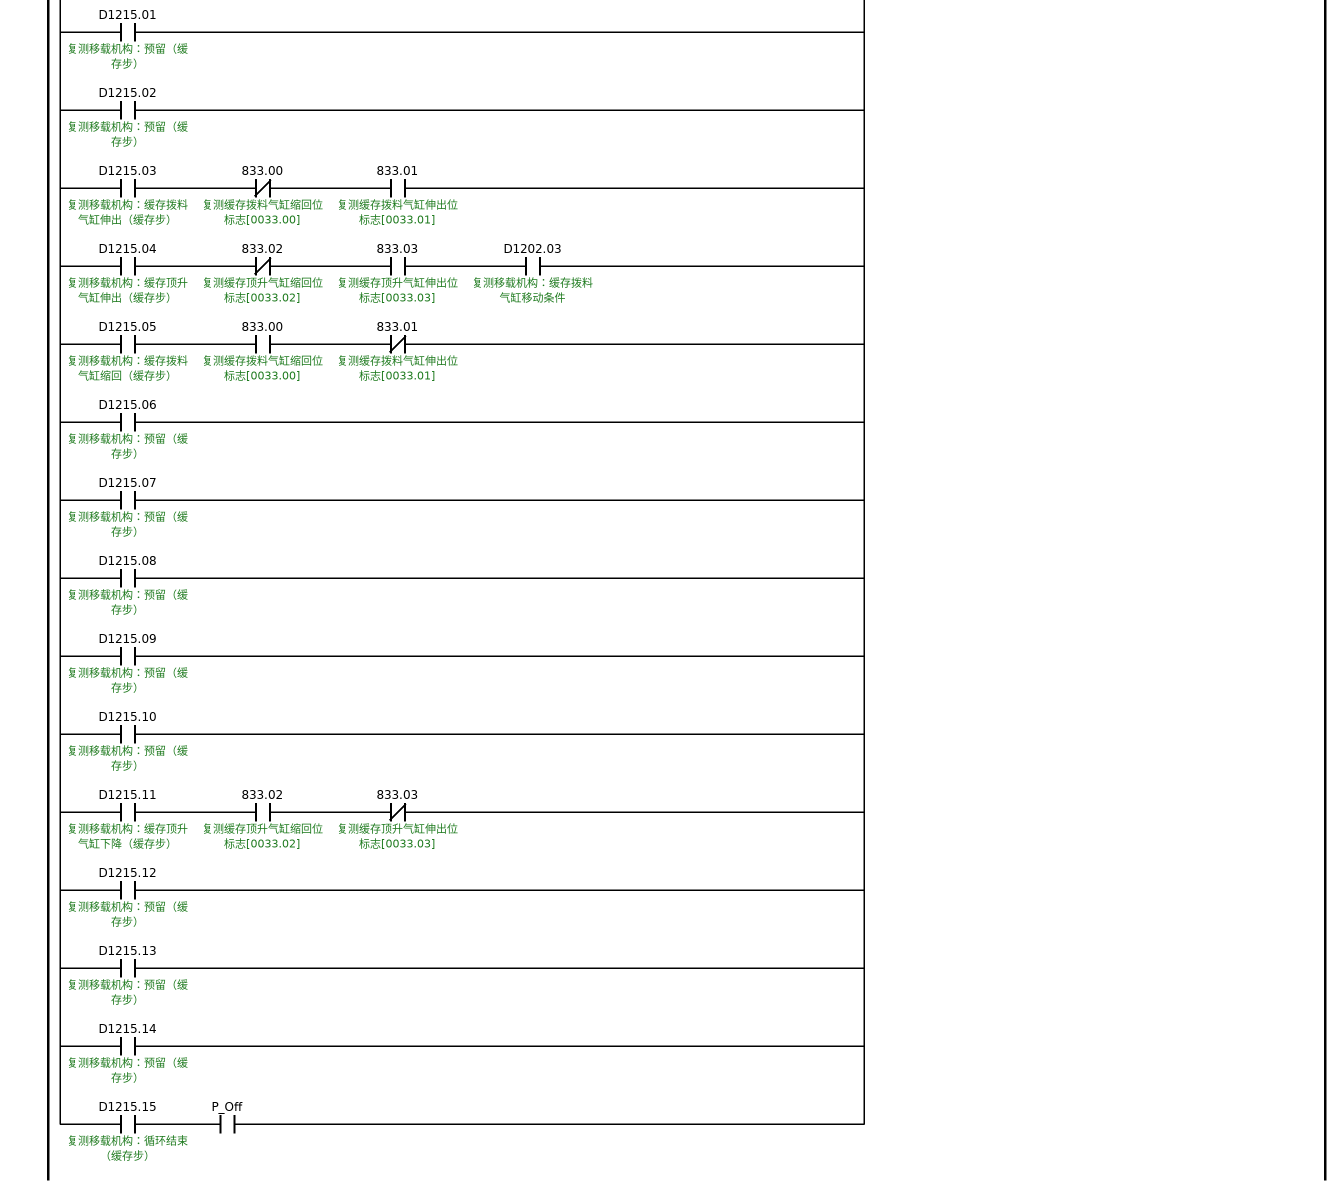
; rung 16: 复测移载机构：步进（缓存步）
LD D1214.00  ; 复测移载机构：自动开始（缓存步）
AND D1205.04  ; 复测移载机构：开始运行条件（缓存步）
AND T1632  ; 复测移栽机构：缓存开始运行延时
OR D1214.01  ; 复测移载机构：预留（缓存步）
LD D1214.02  ; 复测移载机构：判定缓存类型（缓存步）  // 有料执行拨料，无料执行清料（清料跳转至D1215.0）
AND H51.00  ; 复测缓存左1位有料记忆（#1位）
ANDNOT 833.04  ; 复测缓存#1有料感应1标志[0033.04]
AND H51.01  ; 复测缓存右1位有料记忆（#2位）
ANDNOT 833.08  ; 复测缓存#2有料感应1标志[0033.08]
AND D1202.03  ; 复测移载机构：缓存拨料气缸移动条件
ORLD
OR D1214.03  ; 复测移载机构：预留（缓存步）
LD D1214.04  ; 复测移载机构：缓存顶升气缸上升（缓存步）
ANDNOT 833.02  ; 复测缓存顶升气缸缩回位标志[0033.02]
AND 833.03  ; 复测缓存顶升气缸伸出位标志[0033.03]
AND D1202.03  ; 复测移载机构：缓存拨料气缸移动条件
ORLD
LD D1214.05  ; 复测移载机构：缓存拨料气缸伸出（缓存步）
ANDNOT 833.00  ; 复测缓存拨料气缸缩回位标志[0033.00]
AND 833.01  ; 复测缓存拨料气缸伸出位标志[0033.01]
ORLD
OR D1214.06  ; 复测移载机构：预留（缓存步）
OR D1214.07  ; 复测移载机构：预留（缓存步）
OR D1214.08  ; 复测移载机构：预留（缓存步）
OR D1214.09  ; 复测移载机构：预留（缓存步）
LD D1214.10  ; 复测移载机构：缓存顶升气缸下降（缓存步）
AND 833.02  ; 复测缓存顶升气缸缩回位标志[0033.02]
ANDNOT 833.03  ; 复测缓存顶升气缸伸出位标志[0033.03]
ORLD
LD D1214.11  ; 复测移载机构：缓存拨料气缸缩回（缓存步）
AND 833.00  ; 复测缓存拨料气缸缩回位标志[0033.00]
ANDNOT 833.01  ; 复测缓存拨料气缸伸出位标志[0033.01]
ORLD
OR D1214.12  ; 复测移载机构：预留（缓存步）
OR D1214.13  ; 复测移载机构：预留（缓存步）
OR D1214.14  ; 复测移载机构：预留（缓存步）
LD D1214.15  ; 复测移载机构：循环结束（缓存步）
AND P_Off
ORLD
OR D1215.00  ; 复测移载机构：自动开始（缓存步）
OR D1215.01  ; 复测移载机构：预留（缓存步）
OR D1215.02  ; 复测移载机构：预留（缓存步）
LD D1215.03  ; 复测移载机构：缓存拨料气缸伸出（缓存步）
ANDNOT 833.00  ; 复测缓存拨料气缸缩回位标志[0033.00]
AND 833.01  ; 复测缓存拨料气缸伸出位标志[0033.01]
ORLD
LD D1215.04  ; 复测移载机构：缓存顶升气缸伸出（缓存步）
ANDNOT 833.02  ; 复测缓存顶升气缸缩回位标志[0033.02]
AND 833.03  ; 复测缓存顶升气缸伸出位标志[0033.03]
AND D1202.03  ; 复测移载机构：缓存拨料气缸移动条件
ORLD
LD D1215.05  ; 复测移载机构：缓存拨料气缸缩回（缓存步）
AND 833.00  ; 复测缓存拨料气缸缩回位标志[0033.00]
ANDNOT 833.01  ; 复测缓存拨料气缸伸出位标志[0033.01]
ORLD
OR D1215.06  ; 复测移载机构：预留（缓存步）
OR D1215.07  ; 复测移载机构：预留（缓存步）
OR D1215.08  ; 复测移载机构：预留（缓存步）
OR D1215.09  ; 复测移载机构：预留（缓存步）
OR D1215.10  ; 复测移载机构：预留（缓存步）
LD D1215.11  ; 复测移载机构：缓存顶升气缸下降（缓存步）
AND 833.02  ; 复测缓存顶升气缸缩回位标志[0033.02]
ANDNOT 833.03  ; 复测缓存顶升气缸伸出位标志[0033.03]
ORLD
OR D1215.12  ; 复测移载机构：预留（缓存步）
OR D1215.13  ; 复测移载机构：预留（缓存步）
OR D1215.14  ; 复测移载机构：预留（缓存步）
LD D1215.15  ; 复测移载机构：循环结束（缓存步）
AND P_Off
ORLD
LD D1204.00  ; 复测移载机构：单步运行中
@AND D1203.15  ; 复测移载机构：单步（SW）
OR D1204.01  ; 复测移载机构：单步/自动循环运行中（取/放待测料步）
ANDLD
OUT D1205.05  ; $?St$Bk?_#[185] / 复测移载机构：步进条件（缓存步） / $?St$Bk?_#[185]

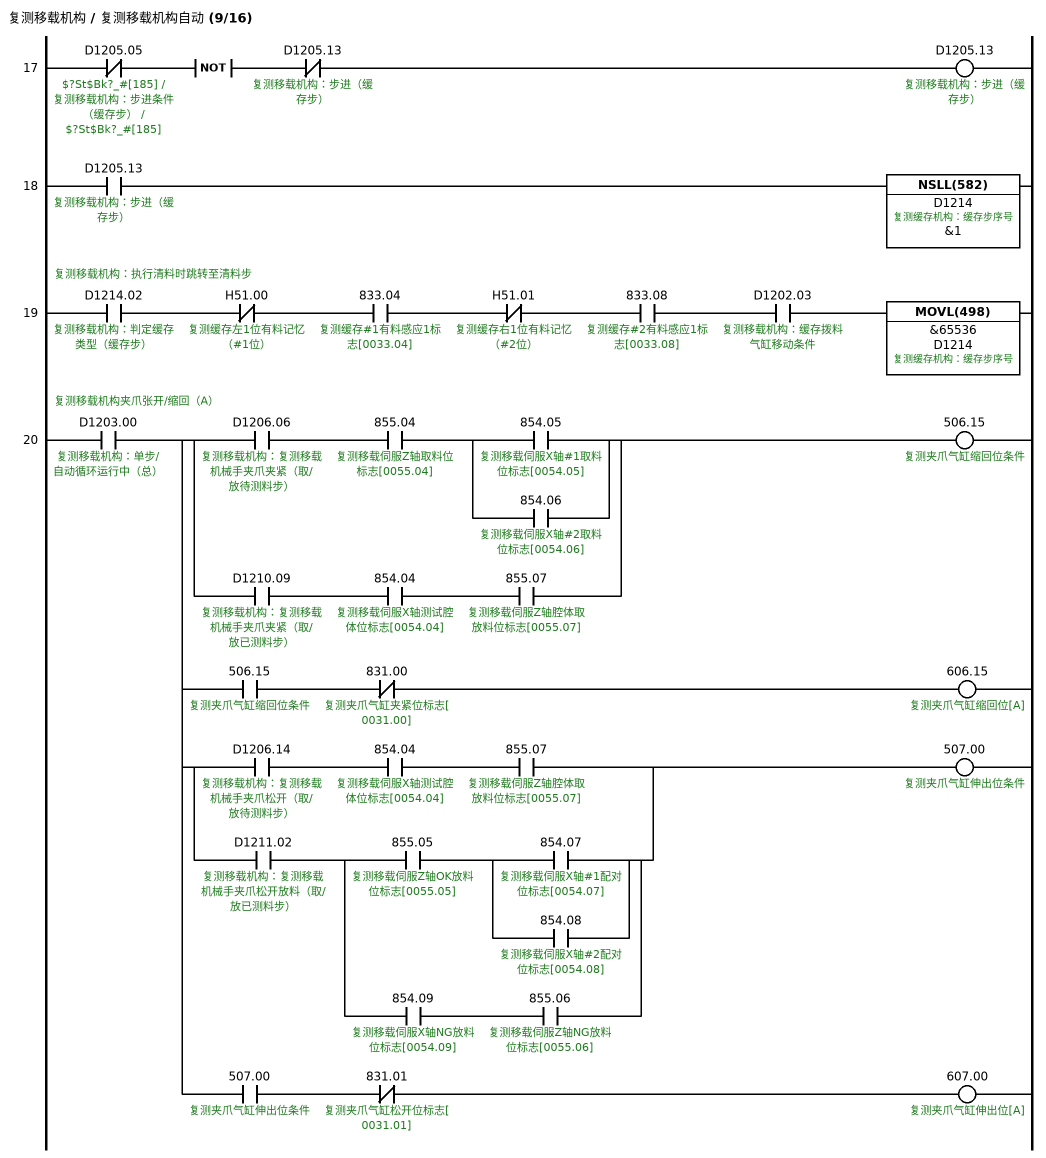
; rung 17
LDNOT D1205.05  ; $?St$Bk?_#[185] / 复测移载机构：步进条件（缓存步） / $?St$Bk?_#[185]
NOT(520)
ANDNOT D1205.13  ; 复测移载机构：步进（缓存步）
OUT D1205.13  ; 复测移载机构：步进（缓存步）
; rung 18
LD D1205.13  ; 复测移载机构：步进（缓存步）
NSLL(582) D1214 &1  ; 复测缓存机构：缓存步序号
; rung 19: 复测移载机构：执行清料时跳转至清料步
LD D1214.02  ; 复测移载机构：判定缓存类型（缓存步）  // 有料执行拨料，无料执行清料（清料跳转至D1215.0）
ANDNOT H51.00  ; 复测缓存左1位有料记忆（#1位）
AND 833.04  ; 复测缓存#1有料感应1标志[0033.04]
ANDNOT H51.01  ; 复测缓存右1位有料记忆（#2位）
AND 833.08  ; 复测缓存#2有料感应1标志[0033.08]
AND D1202.03  ; 复测移载机构：缓存拨料气缸移动条件
MOVL(498) &65536 D1214  ; 复测缓存机构：缓存步序号
; rung 20: 复测移载机构夹爪张开/缩回（A）
LD D1203.00  ; 复测移载机构：单步/自动循环运行中（总）
OUT TR0
LD D1206.06  ; 复测移载机构：复测移载机械手夹爪夹紧（取/放待测料步）
AND 855.04  ; 复测移载伺服Z轴取料位标志[0055.04]
LD 854.05  ; 复测移载伺服X轴#1取料位标志[0054.05]
OR 854.06  ; 复测移载伺服X轴#2取料位标志[0054.06]
ANDLD
LD D1210.09  ; 复测移载机构：复测移载机械手夹爪夹紧（取/放已测料步）
AND 854.04  ; 复测移载伺服X轴测试腔体位标志[0054.04]
AND 855.07  ; 复测移载伺服Z轴腔体取放料位标志[0055.07]
ORLD
ANDLD
OUT 506.15  ; 复测夹爪气缸缩回位条件
LD TR0
AND 506.15  ; 复测夹爪气缸缩回位条件
ANDNOT 831.00  ; 复测夹爪气缸夹紧位标志[0031.00]
OUT 606.15  ; 复测夹爪气缸缩回位[A]
LD TR0
LD D1206.14  ; 复测移载机构：复测移载机械手夹爪松开（取/放待测料步）
AND 854.04  ; 复测移载伺服X轴测试腔体位标志[0054.04]
AND 855.07  ; 复测移载伺服Z轴腔体取放料位标志[0055.07]
LD D1211.02  ; 复测移载机构：复测移载机械手夹爪松开放料（取/放已测料步）
LD 855.05  ; 复测移载伺服Z轴OK放料位标志[0055.05]
LD 854.07  ; 复测移载伺服X轴#1配对位标志[0054.07]
OR 854.08  ; 复测移载伺服X轴#2配对位标志[0054.08]
ANDLD
LD 854.09  ; 复测移载伺服X轴NG放料位标志[0054.09]
AND 855.06  ; 复测移载伺服Z轴NG放料位标志[0055.06]
ORLD
ANDLD
ORLD
ANDLD
OUT 507.00  ; 复测夹爪气缸伸出位条件
LD TR0
AND 507.00  ; 复测夹爪气缸伸出位条件
ANDNOT 831.01  ; 复测夹爪气缸松开位标志[0031.01]
OUT 607.00  ; 复测夹爪气缸伸出位[A]

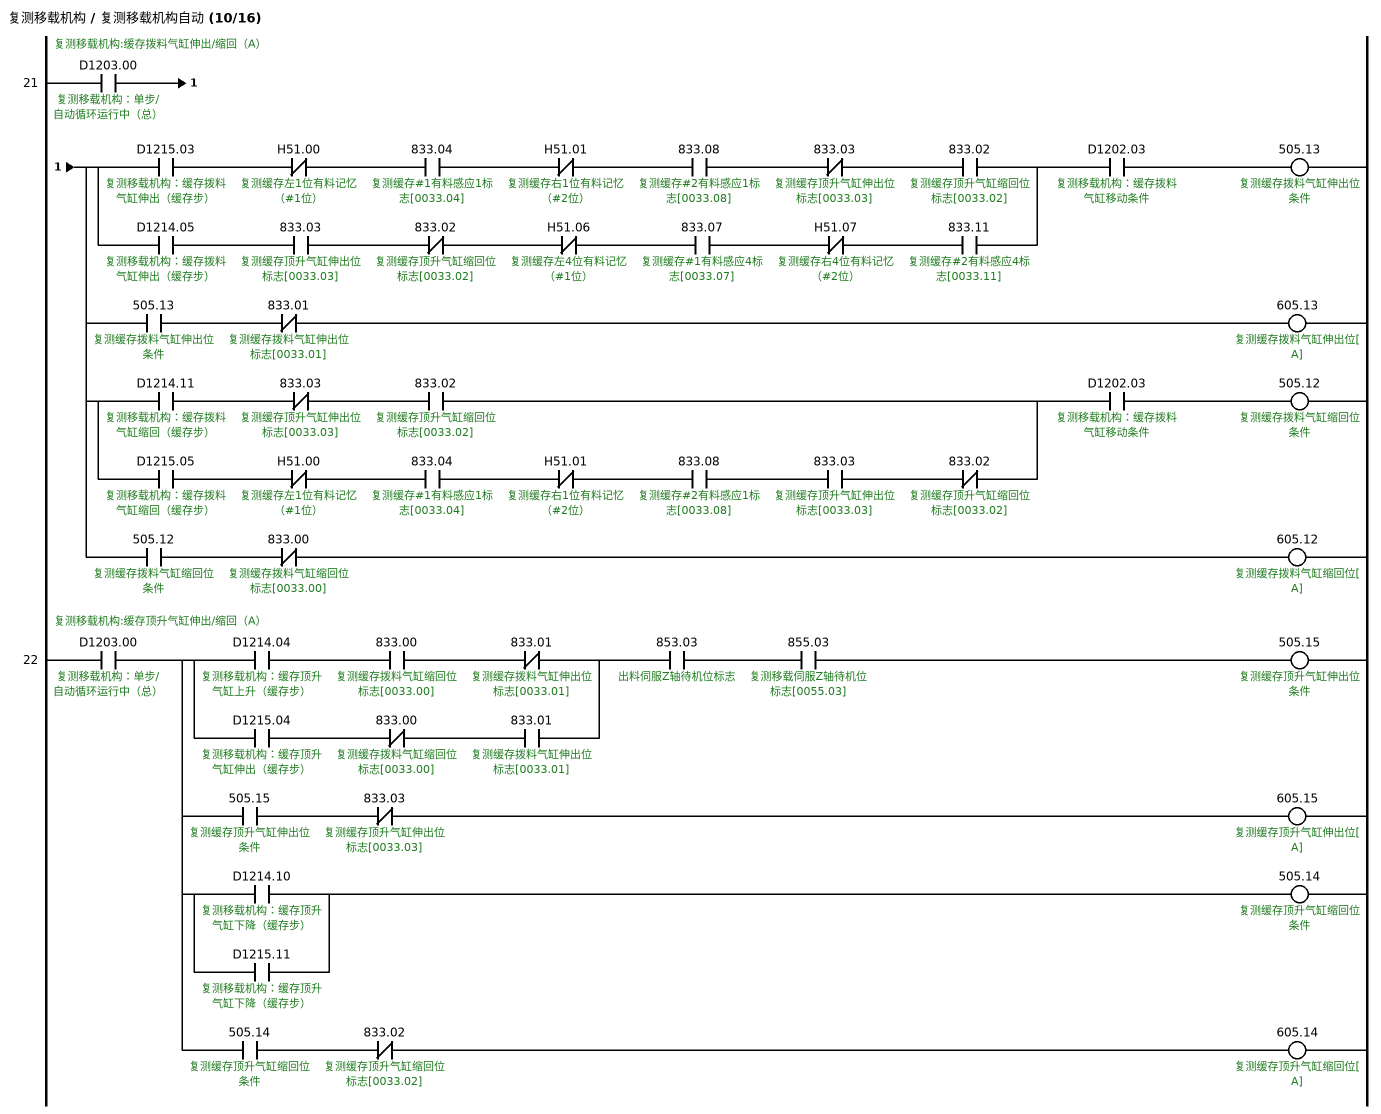
; rung 21: 复测移载机构:缓存拨料气缸伸出/缩回（A）
LD D1203.00  ; 复测移载机构：单步/自动循环运行中（总）
OUT TR0
LD D1215.03  ; 复测移载机构：缓存拨料气缸伸出（缓存步）
ANDNOT H51.00  ; 复测缓存左1位有料记忆（#1位）
AND 833.04  ; 复测缓存#1有料感应1标志[0033.04]
ANDNOT H51.01  ; 复测缓存右1位有料记忆（#2位）
AND 833.08  ; 复测缓存#2有料感应1标志[0033.08]
ANDNOT 833.03  ; 复测缓存顶升气缸伸出位标志[0033.03]
AND 833.02  ; 复测缓存顶升气缸缩回位标志[0033.02]
LD D1214.05  ; 复测移载机构：缓存拨料气缸伸出（缓存步）
AND 833.03  ; 复测缓存顶升气缸伸出位标志[0033.03]
ANDNOT 833.02  ; 复测缓存顶升气缸缩回位标志[0033.02]
ANDNOT H51.06  ; 复测缓存左4位有料记忆（#1位）
AND 833.07  ; 复测缓存#1有料感应4标志[0033.07]
ANDNOT H51.07  ; 复测缓存右4位有料记忆（#2位）
AND 833.11  ; 复测缓存#2有料感应4标志[0033.11]
ORLD
ANDLD
AND D1202.03  ; 复测移载机构：缓存拨料气缸移动条件
OUT 505.13  ; 复测缓存拨料气缸伸出位条件
LD TR0
AND 505.13  ; 复测缓存拨料气缸伸出位条件
ANDNOT 833.01  ; 复测缓存拨料气缸伸出位标志[0033.01]
OUT 605.13  ; 复测缓存拨料气缸伸出位[A]
LD TR0
LD D1214.11  ; 复测移载机构：缓存拨料气缸缩回（缓存步）
ANDNOT 833.03  ; 复测缓存顶升气缸伸出位标志[0033.03]
AND 833.02  ; 复测缓存顶升气缸缩回位标志[0033.02]
LD D1215.05  ; 复测移载机构：缓存拨料气缸缩回（缓存步）
ANDNOT H51.00  ; 复测缓存左1位有料记忆（#1位）
AND 833.04  ; 复测缓存#1有料感应1标志[0033.04]
ANDNOT H51.01  ; 复测缓存右1位有料记忆（#2位）
AND 833.08  ; 复测缓存#2有料感应1标志[0033.08]
AND 833.03  ; 复测缓存顶升气缸伸出位标志[0033.03]
ANDNOT 833.02  ; 复测缓存顶升气缸缩回位标志[0033.02]
ORLD
ANDLD
AND D1202.03  ; 复测移载机构：缓存拨料气缸移动条件
OUT 505.12  ; 复测缓存拨料气缸缩回位条件
LD TR0
AND 505.12  ; 复测缓存拨料气缸缩回位条件
ANDNOT 833.00  ; 复测缓存拨料气缸缩回位标志[0033.00]
OUT 605.12  ; 复测缓存拨料气缸缩回位[A]
; rung 22: 复测移载机构:缓存顶升气缸伸出/缩回（A）
LD D1203.00  ; 复测移载机构：单步/自动循环运行中（总）
OUT TR0
LD D1214.04  ; 复测移载机构：缓存顶升气缸上升（缓存步）
AND 833.00  ; 复测缓存拨料气缸缩回位标志[0033.00]
ANDNOT 833.01  ; 复测缓存拨料气缸伸出位标志[0033.01]
LD D1215.04  ; 复测移载机构：缓存顶升气缸伸出（缓存步）
ANDNOT 833.00  ; 复测缓存拨料气缸缩回位标志[0033.00]
AND 833.01  ; 复测缓存拨料气缸伸出位标志[0033.01]
ORLD
ANDLD
AND 853.03  ; 出料伺服Z轴待机位标志
AND 855.03  ; 复测移载伺服Z轴待机位标志[0055.03]
OUT 505.15  ; 复测缓存顶升气缸伸出位条件
LD TR0
AND 505.15  ; 复测缓存顶升气缸伸出位条件
ANDNOT 833.03  ; 复测缓存顶升气缸伸出位标志[0033.03]
OUT 605.15  ; 复测缓存顶升气缸伸出位[A]
LD TR0
LD D1214.10  ; 复测移载机构：缓存顶升气缸下降（缓存步）
OR D1215.11  ; 复测移载机构：缓存顶升气缸下降（缓存步）
ANDLD
OUT 505.14  ; 复测缓存顶升气缸缩回位条件
LD TR0
AND 505.14  ; 复测缓存顶升气缸缩回位条件
ANDNOT 833.02  ; 复测缓存顶升气缸缩回位标志[0033.02]
OUT 605.14  ; 复测缓存顶升气缸缩回位[A]

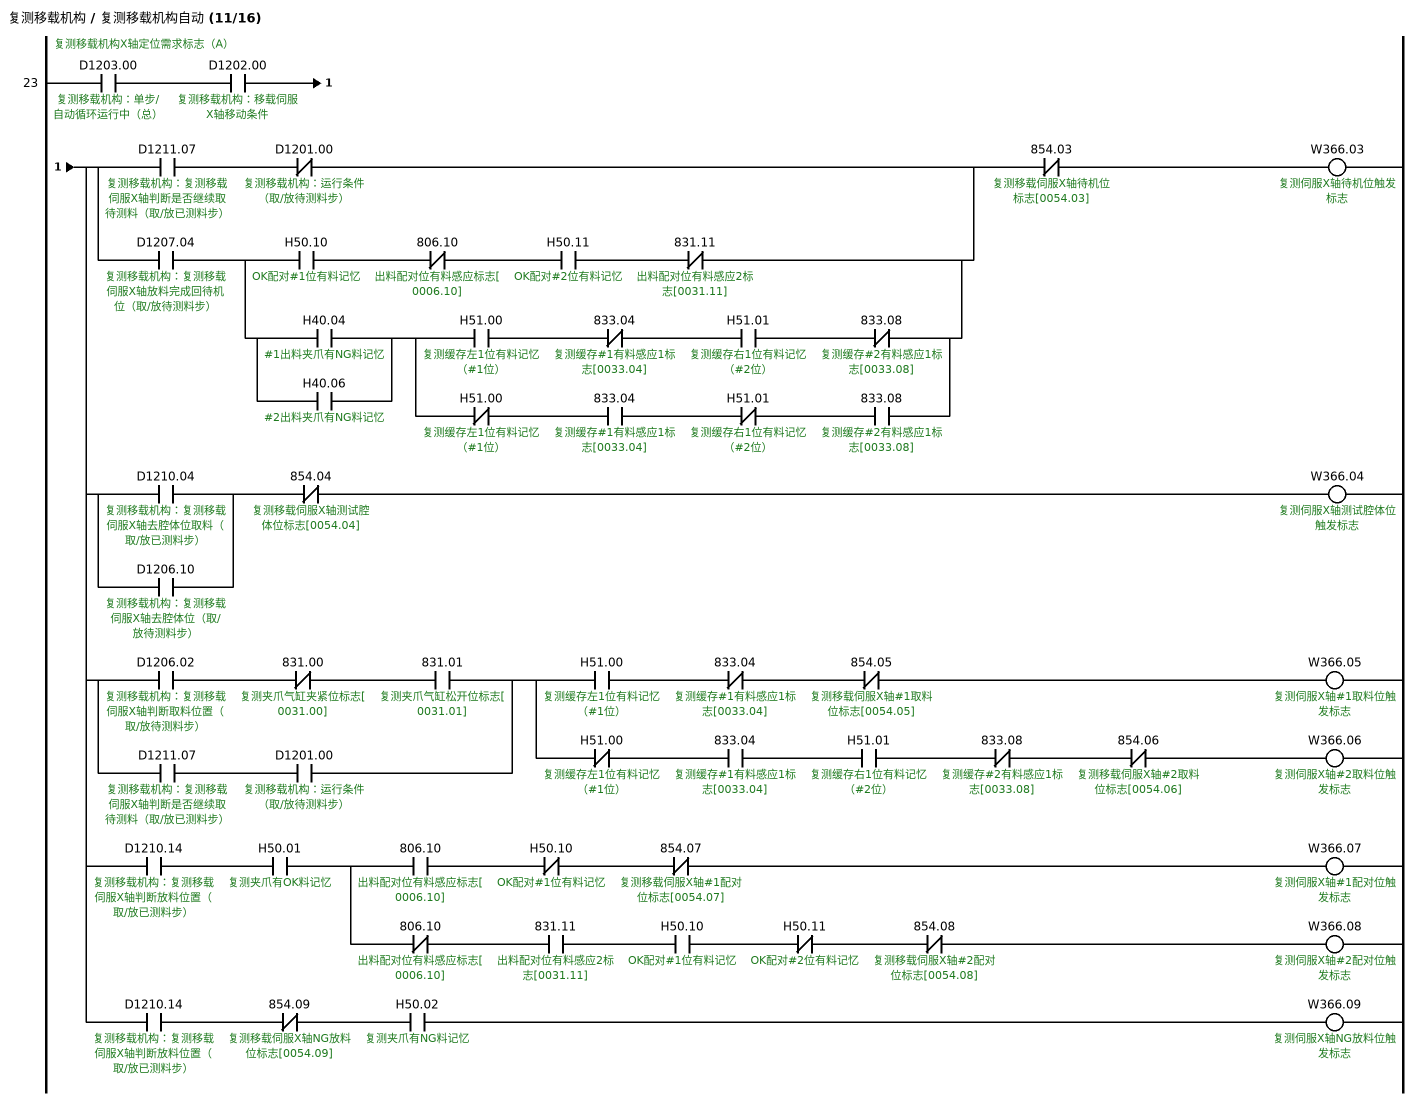
; rung 23: 复测移载机构X轴定位需求标志（A）
LD D1203.00  ; 复测移载机构：单步/自动循环运行中（总）
AND D1202.00  ; 复测移载机构：移载伺服X轴移动条件
OUT TR0
LD D1211.07  ; 复测移载机构：复测移载伺服X轴判断是否继续取待测料（取/放已测料步）
ANDNOT D1201.00  ; 复测移载机构：运行条件（取/放待测料步）
LD D1207.04  ; 复测移载机构：复测移载伺服X轴放料完成回待机位（取/放待测料步）
LD H50.10  ; OK配对#1位有料记忆
ANDNOT 806.10  ; 出料配对位有料感应标志[0006.10]
AND H50.11  ; OK配对#2位有料记忆
ANDNOT 831.11  ; 出料配对位有料感应2标志[0031.11]
LD H40.04  ; #1出料夹爪有NG料记忆
OR H40.06  ; #2出料夹爪有NG料记忆
LD H51.00  ; 复测缓存左1位有料记忆（#1位）
ANDNOT 833.04  ; 复测缓存#1有料感应1标志[0033.04]
AND H51.01  ; 复测缓存右1位有料记忆（#2位）
ANDNOT 833.08  ; 复测缓存#2有料感应1标志[0033.08]
LDNOT H51.00  ; 复测缓存左1位有料记忆（#1位）
AND 833.04  ; 复测缓存#1有料感应1标志[0033.04]
ANDNOT H51.01  ; 复测缓存右1位有料记忆（#2位）
AND 833.08  ; 复测缓存#2有料感应1标志[0033.08]
ORLD
ANDLD
ORLD
ANDLD
ORLD
ANDLD
ANDNOT 854.03  ; 复测移载伺服X轴待机位标志[0054.03]
OUT W366.03  ; 复测伺服X轴待机位触发标志
LD TR0
LD D1210.04  ; 复测移载机构：复测移载伺服X轴去腔体位取料（取/放已测料步）
OR D1206.10  ; 复测移载机构：复测移载伺服X轴去腔体位（取/放待测料步）
ANDLD
ANDNOT 854.04  ; 复测移载伺服X轴测试腔体位标志[0054.04]
OUT W366.04  ; 复测伺服X轴测试腔体位触发标志
LD TR0
LD D1206.02  ; 复测移载机构：复测移载伺服X轴判断取料位置（取/放待测料步）
ANDNOT 831.00  ; 复测夹爪气缸夹紧位标志[0031.00]
AND 831.01  ; 复测夹爪气缸松开位标志[0031.01]
LD D1211.07  ; 复测移载机构：复测移载伺服X轴判断是否继续取待测料（取/放已测料步）
AND D1201.00  ; 复测移载机构：运行条件（取/放待测料步）
ORLD
ANDLD
OUT TR1
AND H51.00  ; 复测缓存左1位有料记忆（#1位）
ANDNOT 833.04  ; 复测缓存#1有料感应1标志[0033.04]
ANDNOT 854.05  ; 复测移载伺服X轴#1取料位标志[0054.05]
OUT W366.05  ; 复测伺服X轴#1取料位触发标志
LD TR1
ANDNOT H51.00  ; 复测缓存左1位有料记忆（#1位）
AND 833.04  ; 复测缓存#1有料感应1标志[0033.04]
AND H51.01  ; 复测缓存右1位有料记忆（#2位）
ANDNOT 833.08  ; 复测缓存#2有料感应1标志[0033.08]
ANDNOT 854.06  ; 复测移载伺服X轴#2取料位标志[0054.06]
OUT W366.06  ; 复测伺服X轴#2取料位触发标志
LD TR0
AND D1210.14  ; 复测移载机构：复测移载伺服X轴判断放料位置（取/放已测料步）
AND H50.01  ; 复测夹爪有OK料记忆
OUT TR1
AND 806.10  ; 出料配对位有料感应标志[0006.10]
ANDNOT H50.10  ; OK配对#1位有料记忆
ANDNOT 854.07  ; 复测移载伺服X轴#1配对位标志[0054.07]
OUT W366.07  ; 复测伺服X轴#1配对位触发标志
LD TR1
ANDNOT 806.10  ; 出料配对位有料感应标志[0006.10]
AND 831.11  ; 出料配对位有料感应2标志[0031.11]
AND H50.10  ; OK配对#1位有料记忆
ANDNOT H50.11  ; OK配对#2位有料记忆
ANDNOT 854.08  ; 复测移载伺服X轴#2配对位标志[0054.08]
OUT W366.08  ; 复测伺服X轴#2配对位触发标志
LD TR0
AND D1210.14  ; 复测移载机构：复测移载伺服X轴判断放料位置（取/放已测料步）
ANDNOT 854.09  ; 复测移载伺服X轴NG放料位标志[0054.09]
AND H50.02  ; 复测夹爪有NG料记忆
OUT W366.09  ; 复测伺服X轴NG放料位触发标志

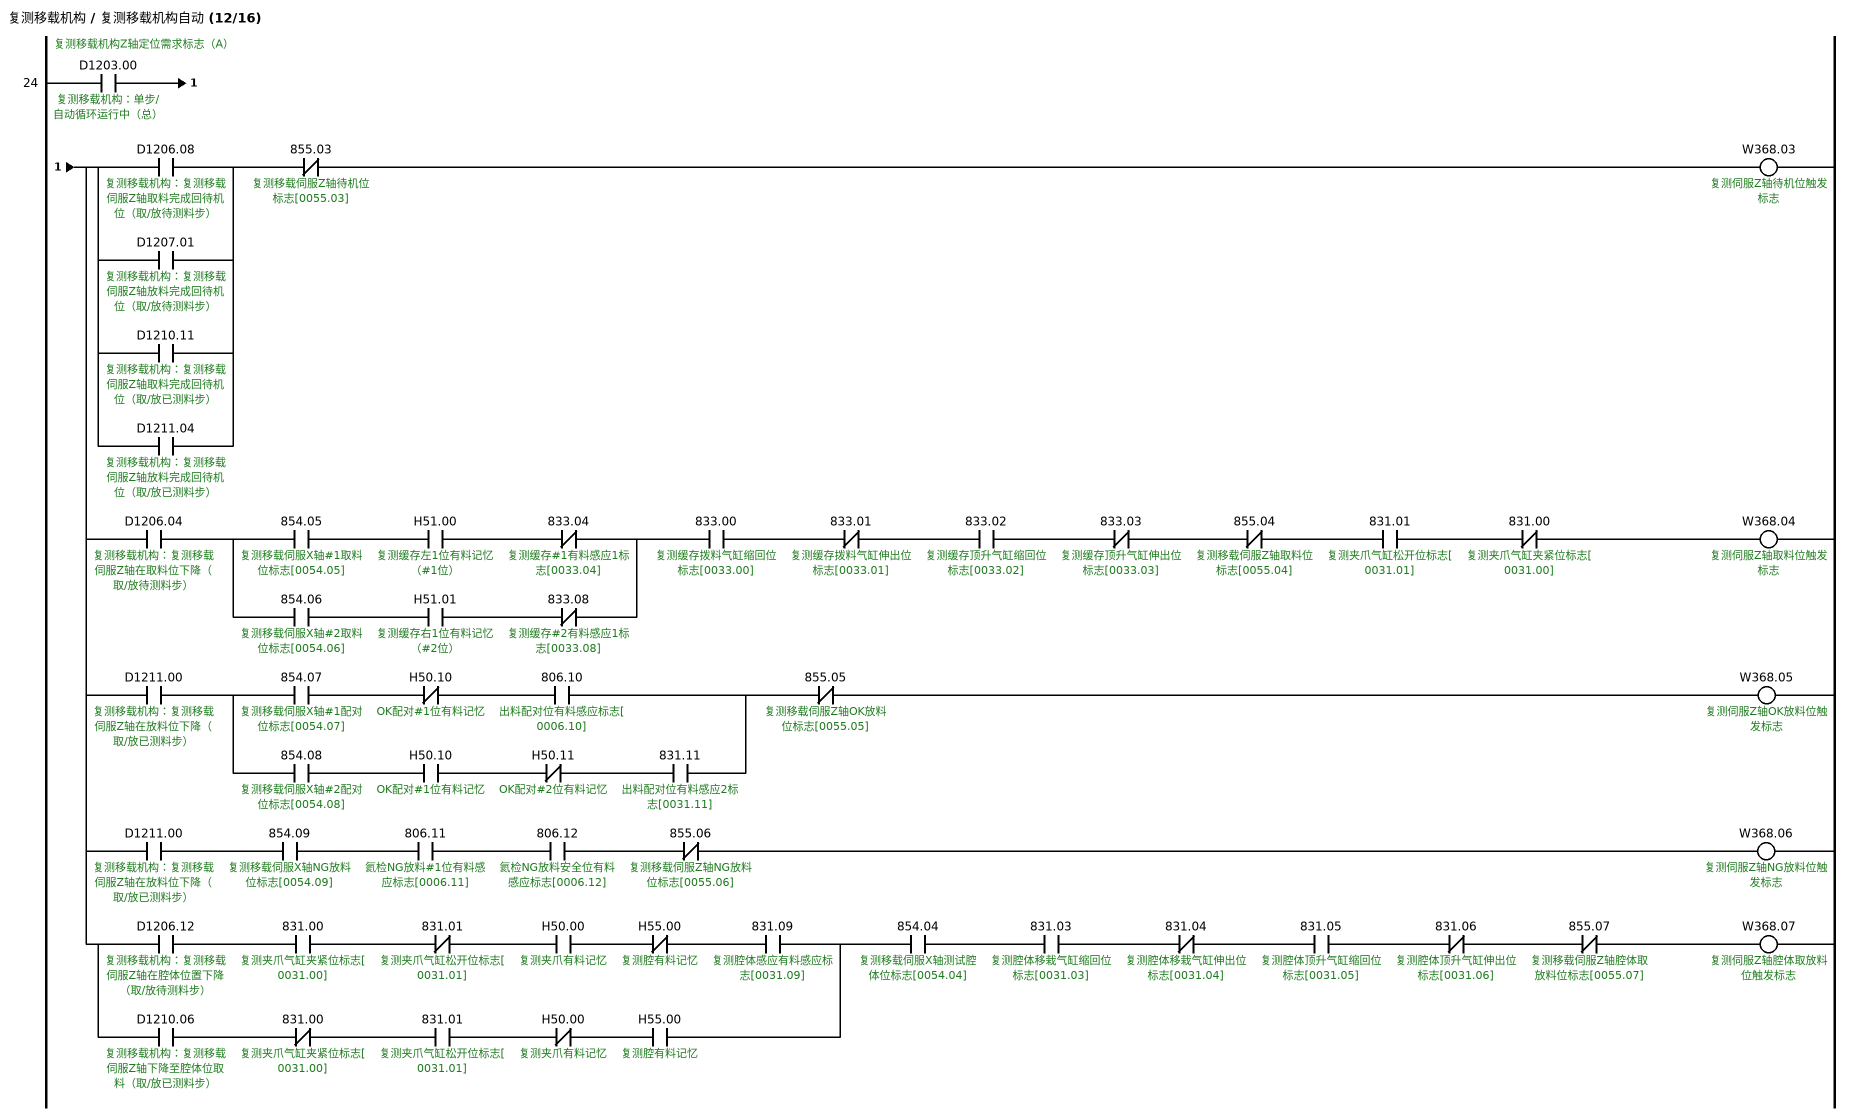
; rung 24: 复测移载机构Z轴定位需求标志（A）
LD D1203.00  ; 复测移载机构：单步/自动循环运行中（总）
OUT TR0
LD D1206.08  ; 复测移载机构：复测移载伺服Z轴取料完成回待机位（取/放待测料步）
OR D1207.01  ; 复测移载机构：复测移载伺服Z轴放料完成回待机位（取/放待测料步）
OR D1210.11  ; 复测移载机构：复测移载伺服Z轴取料完成回待机位（取/放已测料步）
OR D1211.04  ; 复测移载机构：复测移载伺服Z轴放料完成回待机位（取/放已测料步）
ANDLD
ANDNOT 855.03  ; 复测移载伺服Z轴待机位标志[0055.03]
OUT W368.03  ; 复测伺服Z轴待机位触发标志
LD TR0
AND D1206.04  ; 复测移载机构：复测移载伺服Z轴在取料位下降（取/放待测料步）
LD 854.05  ; 复测移载伺服X轴#1取料位标志[0054.05]
AND H51.00  ; 复测缓存左1位有料记忆（#1位）
ANDNOT 833.04  ; 复测缓存#1有料感应1标志[0033.04]
LD 854.06  ; 复测移载伺服X轴#2取料位标志[0054.06]
AND H51.01  ; 复测缓存右1位有料记忆（#2位）
ANDNOT 833.08  ; 复测缓存#2有料感应1标志[0033.08]
ORLD
ANDLD
AND 833.00  ; 复测缓存拨料气缸缩回位标志[0033.00]
ANDNOT 833.01  ; 复测缓存拨料气缸伸出位标志[0033.01]
AND 833.02  ; 复测缓存顶升气缸缩回位标志[0033.02]
ANDNOT 833.03  ; 复测缓存顶升气缸伸出位标志[0033.03]
ANDNOT 855.04  ; 复测移载伺服Z轴取料位标志[0055.04]
AND 831.01  ; 复测夹爪气缸松开位标志[0031.01]
ANDNOT 831.00  ; 复测夹爪气缸夹紧位标志[0031.00]
OUT W368.04  ; 复测伺服Z轴取料位触发标志
LD TR0
AND D1211.00  ; 复测移载机构：复测移载伺服Z轴在放料位下降（取/放已测料步）
LD 854.07  ; 复测移载伺服X轴#1配对位标志[0054.07]
ANDNOT H50.10  ; OK配对#1位有料记忆
AND 806.10  ; 出料配对位有料感应标志[0006.10]
LD 854.08  ; 复测移载伺服X轴#2配对位标志[0054.08]
AND H50.10  ; OK配对#1位有料记忆
ANDNOT H50.11  ; OK配对#2位有料记忆
AND 831.11  ; 出料配对位有料感应2标志[0031.11]
ORLD
ANDLD
ANDNOT 855.05  ; 复测移载伺服Z轴OK放料位标志[0055.05]
OUT W368.05  ; 复测伺服Z轴OK放料位触发标志
LD TR0
AND D1211.00  ; 复测移载机构：复测移载伺服Z轴在放料位下降（取/放已测料步）
AND 854.09  ; 复测移载伺服X轴NG放料位标志[0054.09]
AND 806.11  ; 氦检NG放料#1位有料感应标志[0006.11]
AND 806.12  ; 氦检NG放料安全位有料感应标志[0006.12]
ANDNOT 855.06  ; 复测移载伺服Z轴NG放料位标志[0055.06]
OUT W368.06  ; 复测伺服Z轴NG放料位触发标志
LD TR0
LD D1206.12  ; 复测移载机构：复测移载伺服Z轴在腔体位置下降（取/放待测料步）
AND 831.00  ; 复测夹爪气缸夹紧位标志[0031.00]
ANDNOT 831.01  ; 复测夹爪气缸松开位标志[0031.01]
AND H50.00  ; 复测夹爪有料记忆
ANDNOT H55.00  ; 复测腔有料记忆
AND 831.09  ; 复测腔体感应有料感应标志[0031.09]
LD D1210.06  ; 复测移载机构：复测移载伺服Z轴下降至腔体位取料（取/放已测料步）
ANDNOT 831.00  ; 复测夹爪气缸夹紧位标志[0031.00]
AND 831.01  ; 复测夹爪气缸松开位标志[0031.01]
ANDNOT H50.00  ; 复测夹爪有料记忆
AND H55.00  ; 复测腔有料记忆
ORLD
ANDLD
AND 854.04  ; 复测移载伺服X轴测试腔体位标志[0054.04]
AND 831.03  ; 复测腔体移栽气缸缩回位标志[0031.03]
ANDNOT 831.04  ; 复测腔体移栽气缸伸出位标志[0031.04]
AND 831.05  ; 复测腔体顶升气缸缩回位标志[0031.05]
ANDNOT 831.06  ; 复测腔体顶升气缸伸出位标志[0031.06]
ANDNOT 855.07  ; 复测移载伺服Z轴腔体取放料位标志[0055.07]
OUT W368.07  ; 复测伺服Z轴腔体取放料位触发标志

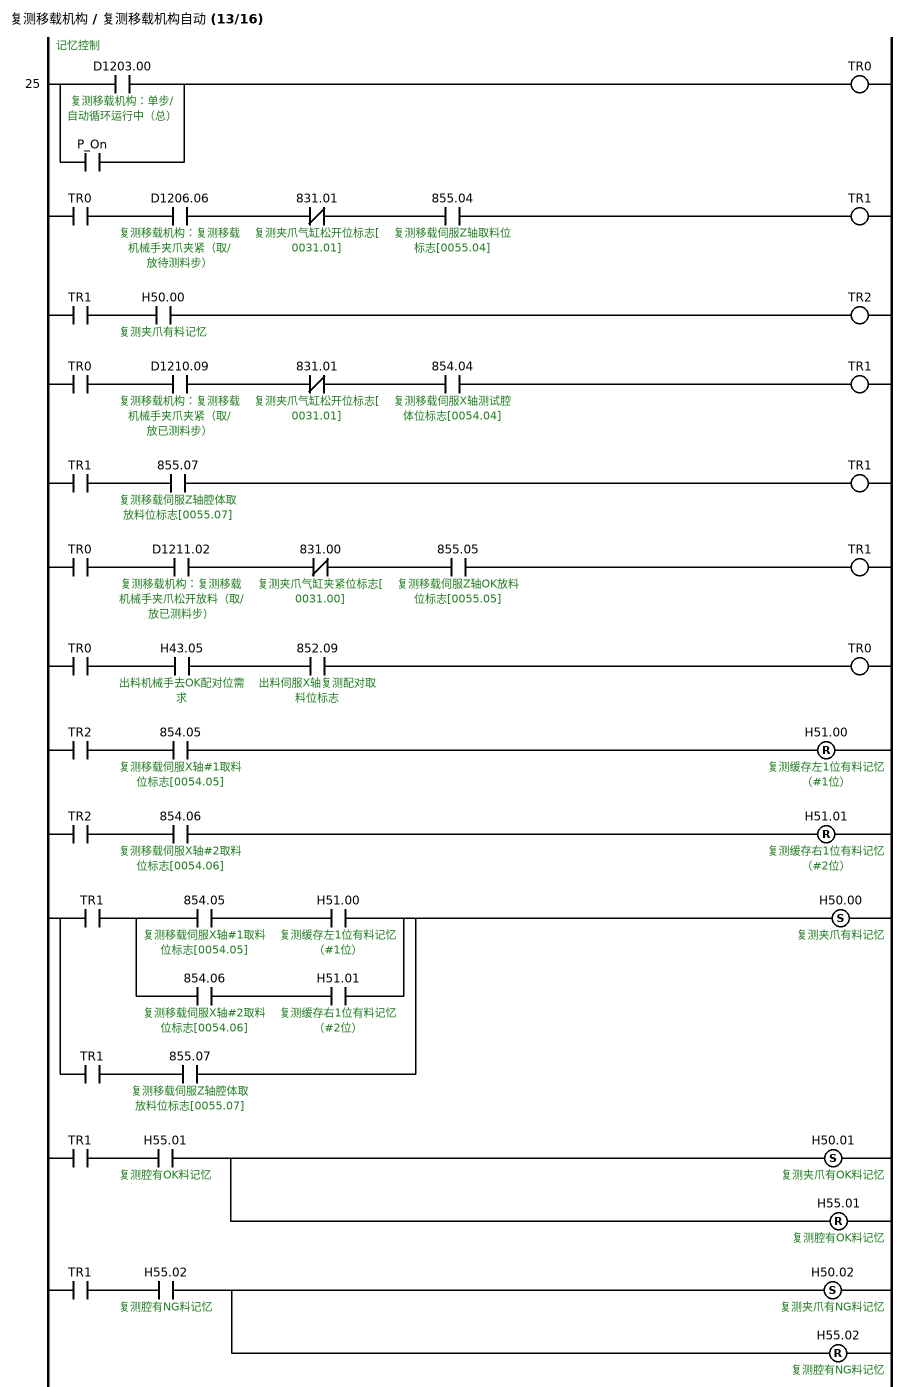

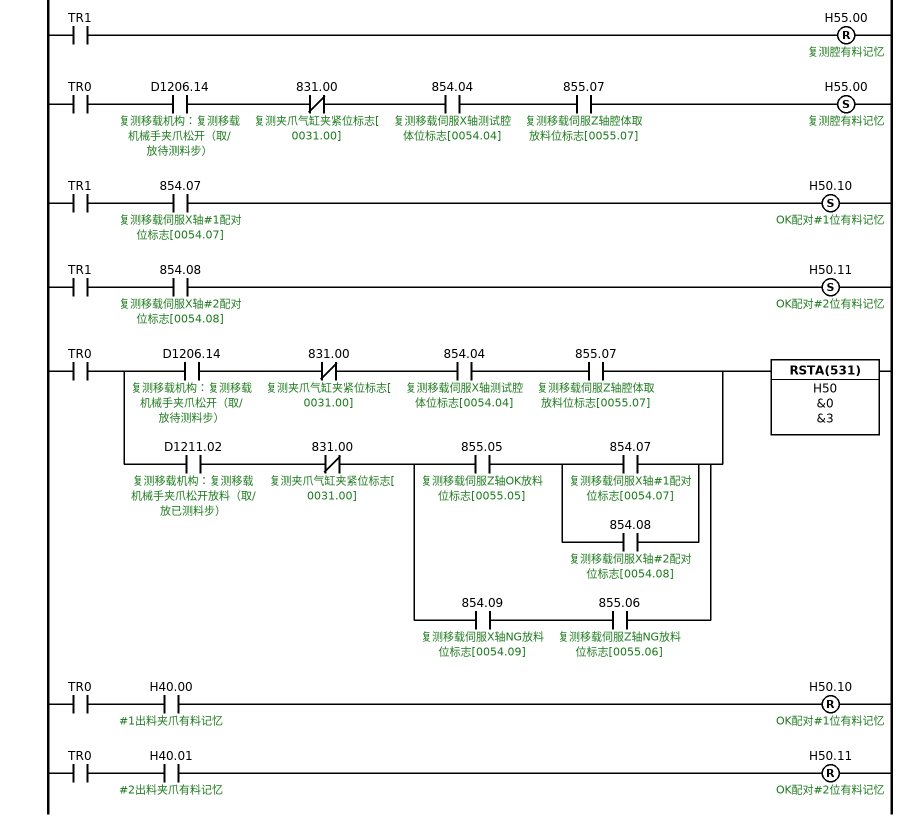
; rung 25: 记忆控制
LD D1203.00  ; 复测移载机构：单步/自动循环运行中（总）
OR P_On
OUT TR0
AND D1206.06  ; 复测移载机构：复测移载机械手夹爪夹紧（取/放待测料步）
ANDNOT 831.01  ; 复测夹爪气缸松开位标志[0031.01]
AND 855.04  ; 复测移载伺服Z轴取料位标志[0055.04]
OUT TR1
AND H50.00  ; 复测夹爪有料记忆
OUT TR2
AND 854.05  ; 复测移载伺服X轴#1取料位标志[0054.05]
RSET H51.00  ; 复测缓存左1位有料记忆（#1位）
LD TR2
AND 854.06  ; 复测移载伺服X轴#2取料位标志[0054.06]
RSET H51.01  ; 复测缓存右1位有料记忆（#2位）
LD TR1
LD 854.05  ; 复测移载伺服X轴#1取料位标志[0054.05]
AND H51.00  ; 复测缓存左1位有料记忆（#1位）
LD 854.06  ; 复测移载伺服X轴#2取料位标志[0054.06]
AND H51.01  ; 复测缓存右1位有料记忆（#2位）
ORLD
ANDLD
LD TR0
AND D1210.09  ; 复测移载机构：复测移载机械手夹爪夹紧（取/放已测料步）
ANDNOT 831.01  ; 复测夹爪气缸松开位标志[0031.01]
AND 854.04  ; 复测移载伺服X轴测试腔体位标志[0054.04]
OUT TR1
AND 855.07  ; 复测移载伺服Z轴腔体取放料位标志[0055.07]
ORLD
SET H50.00  ; 复测夹爪有料记忆
LD TR1
AND 855.07  ; 复测移载伺服Z轴腔体取放料位标志[0055.07]
OUT TR1
AND H55.01  ; 复测腔有OK料记忆
SET H50.01  ; 复测夹爪有OK料记忆
RSET H55.01  ; 复测腔有OK料记忆
LD TR1
AND H55.02  ; 复测腔有NG料记忆
SET H50.02  ; 复测夹爪有NG料记忆
RSET H55.02  ; 复测腔有NG料记忆
LD TR1
RSET H55.00  ; 复测腔有料记忆
LD TR0
AND D1206.14  ; 复测移载机构：复测移载机械手夹爪松开（取/放待测料步）
ANDNOT 831.00  ; 复测夹爪气缸夹紧位标志[0031.00]
AND 854.04  ; 复测移载伺服X轴测试腔体位标志[0054.04]
AND 855.07  ; 复测移载伺服Z轴腔体取放料位标志[0055.07]
SET H55.00  ; 复测腔有料记忆
LD TR0
AND D1211.02  ; 复测移载机构：复测移载机械手夹爪松开放料（取/放已测料步）
ANDNOT 831.00  ; 复测夹爪气缸夹紧位标志[0031.00]
AND 855.05  ; 复测移载伺服Z轴OK放料位标志[0055.05]
OUT TR1
AND 854.07  ; 复测移载伺服X轴#1配对位标志[0054.07]
SET H50.10  ; OK配对#1位有料记忆
LD TR1
AND 854.08  ; 复测移载伺服X轴#2配对位标志[0054.08]
SET H50.11  ; OK配对#2位有料记忆
LD TR0
LD D1206.14  ; 复测移载机构：复测移载机械手夹爪松开（取/放待测料步）
ANDNOT 831.00  ; 复测夹爪气缸夹紧位标志[0031.00]
AND 854.04  ; 复测移载伺服X轴测试腔体位标志[0054.04]
AND 855.07  ; 复测移载伺服Z轴腔体取放料位标志[0055.07]
LD D1211.02  ; 复测移载机构：复测移载机械手夹爪松开放料（取/放已测料步）
ANDNOT 831.00  ; 复测夹爪气缸夹紧位标志[0031.00]
LD 855.05  ; 复测移载伺服Z轴OK放料位标志[0055.05]
LD 854.07  ; 复测移载伺服X轴#1配对位标志[0054.07]
OR 854.08  ; 复测移载伺服X轴#2配对位标志[0054.08]
ANDLD
LD 854.09  ; 复测移载伺服X轴NG放料位标志[0054.09]
AND 855.06  ; 复测移载伺服Z轴NG放料位标志[0055.06]
ORLD
ANDLD
ORLD
ANDLD
RSTA(531) H50 &0 &3
LD TR0
AND H43.05  ; 出料机械手去OK配对位需求
AND 852.09  ; 出料伺服X轴复测配对取料位标志
OUT TR0
AND H40.00  ; #1出料夹爪有料记忆
RSET H50.10  ; OK配对#1位有料记忆
LD TR0
AND H40.01  ; #2出料夹爪有料记忆
RSET H50.11  ; OK配对#2位有料记忆

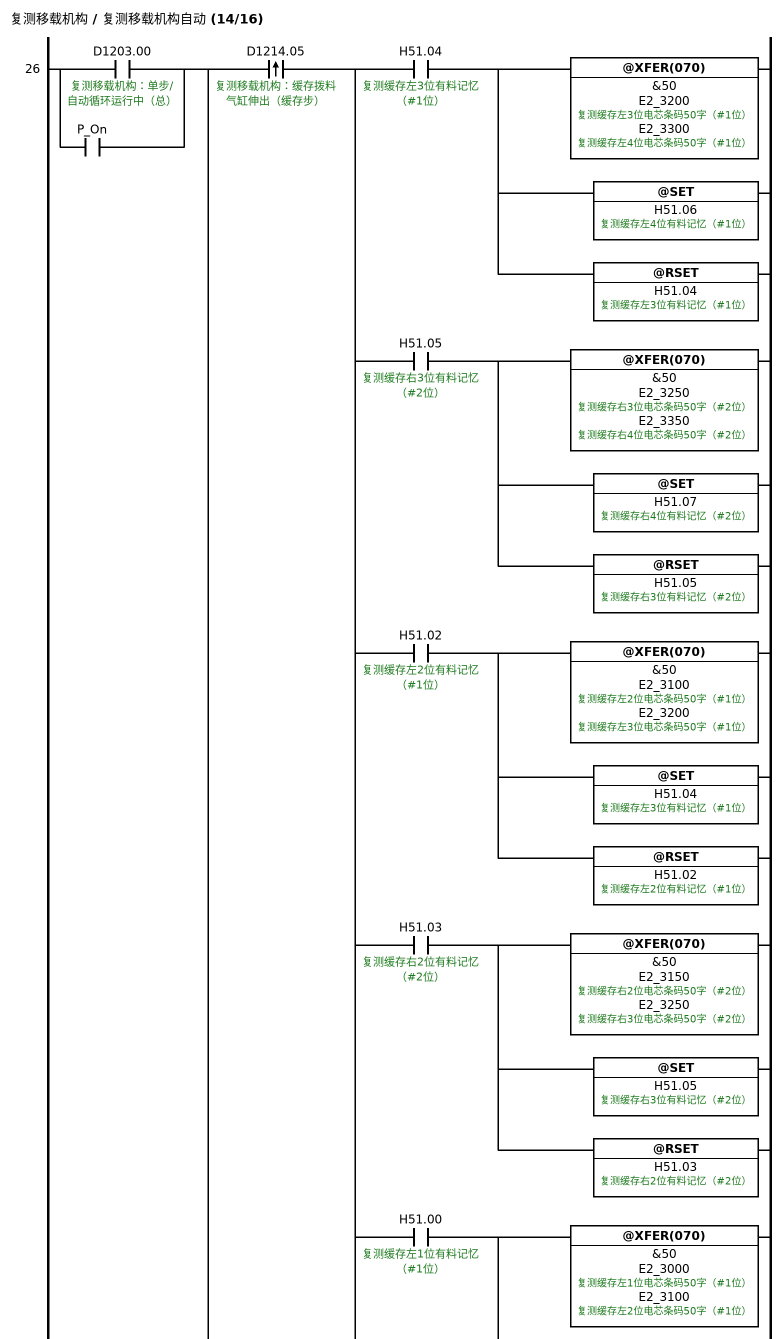

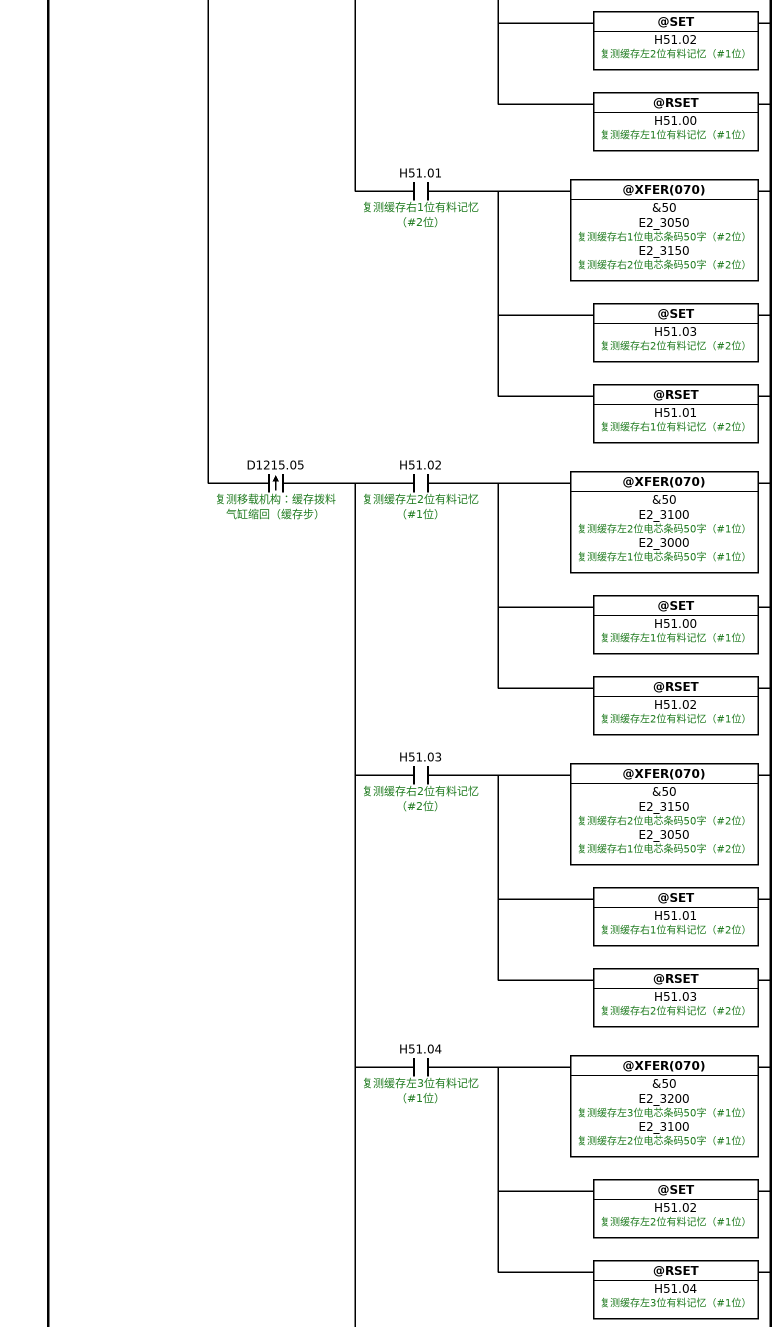

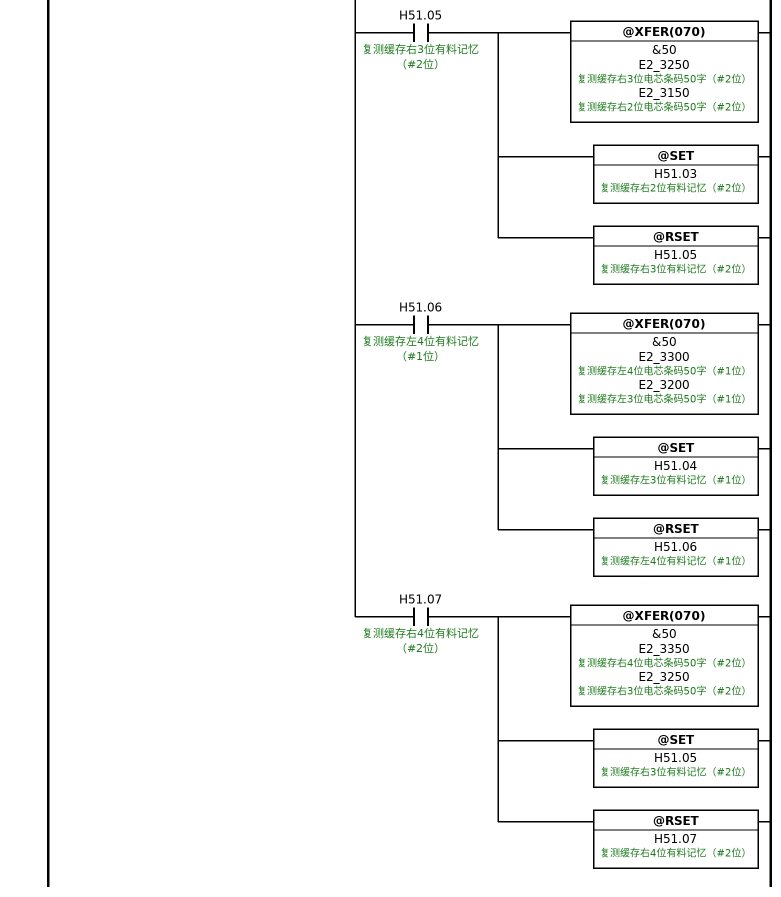
; rung 26
LD D1203.00  ; 复测移载机构：单步/自动循环运行中（总）
OR P_On
OUT TR0
@AND D1214.05  ; 复测移载机构：缓存拨料气缸伸出（缓存步）
OUT TR1
AND H51.04  ; 复测缓存左3位有料记忆（#1位）
@XFER(070) &50 E2_3200 E2_3300  ; 复测缓存左3位电芯条码50字（#1位）, 复测缓存左4位电芯条码50字（#1位）
@SET H51.06  ; 复测缓存左4位有料记忆（#1位）
@RSET H51.04  ; 复测缓存左3位有料记忆（#1位）
LD TR1
AND H51.05  ; 复测缓存右3位有料记忆（#2位）
@XFER(070) &50 E2_3250 E2_3350  ; 复测缓存右3位电芯条码50字（#2位）, 复测缓存右4位电芯条码50字（#2位）
@SET H51.07  ; 复测缓存右4位有料记忆（#2位）
@RSET H51.05  ; 复测缓存右3位有料记忆（#2位）
LD TR1
AND H51.02  ; 复测缓存左2位有料记忆（#1位）
@XFER(070) &50 E2_3100 E2_3200  ; 复测缓存左2位电芯条码50字（#1位）, 复测缓存左3位电芯条码50字（#1位）
@SET H51.04  ; 复测缓存左3位有料记忆（#1位）
@RSET H51.02  ; 复测缓存左2位有料记忆（#1位）
LD TR1
AND H51.03  ; 复测缓存右2位有料记忆（#2位）
@XFER(070) &50 E2_3150 E2_3250  ; 复测缓存右2位电芯条码50字（#2位）, 复测缓存右3位电芯条码50字（#2位）
@SET H51.05  ; 复测缓存右3位有料记忆（#2位）
@RSET H51.03  ; 复测缓存右2位有料记忆（#2位）
LD TR1
AND H51.00  ; 复测缓存左1位有料记忆（#1位）
@XFER(070) &50 E2_3000 E2_3100  ; 复测缓存左1位电芯条码50字（#1位）, 复测缓存左2位电芯条码50字（#1位）
@SET H51.02  ; 复测缓存左2位有料记忆（#1位）
@RSET H51.00  ; 复测缓存左1位有料记忆（#1位）
LD TR1
AND H51.01  ; 复测缓存右1位有料记忆（#2位）
@XFER(070) &50 E2_3050 E2_3150  ; 复测缓存右1位电芯条码50字（#2位）, 复测缓存右2位电芯条码50字（#2位）
@SET H51.03  ; 复测缓存右2位有料记忆（#2位）
@RSET H51.01  ; 复测缓存右1位有料记忆（#2位）
LD TR0
@AND D1215.05  ; 复测移载机构：缓存拨料气缸缩回（缓存步）
OUT TR0
AND H51.02  ; 复测缓存左2位有料记忆（#1位）
@XFER(070) &50 E2_3100 E2_3000  ; 复测缓存左2位电芯条码50字（#1位）, 复测缓存左1位电芯条码50字（#1位）
@SET H51.00  ; 复测缓存左1位有料记忆（#1位）
@RSET H51.02  ; 复测缓存左2位有料记忆（#1位）
LD TR0
AND H51.03  ; 复测缓存右2位有料记忆（#2位）
@XFER(070) &50 E2_3150 E2_3050  ; 复测缓存右2位电芯条码50字（#2位）, 复测缓存右1位电芯条码50字（#2位）
@SET H51.01  ; 复测缓存右1位有料记忆（#2位）
@RSET H51.03  ; 复测缓存右2位有料记忆（#2位）
LD TR0
AND H51.04  ; 复测缓存左3位有料记忆（#1位）
@XFER(070) &50 E2_3200 E2_3100  ; 复测缓存左3位电芯条码50字（#1位）, 复测缓存左2位电芯条码50字（#1位）
@SET H51.02  ; 复测缓存左2位有料记忆（#1位）
@RSET H51.04  ; 复测缓存左3位有料记忆（#1位）
LD TR0
AND H51.05  ; 复测缓存右3位有料记忆（#2位）
@XFER(070) &50 E2_3250 E2_3150  ; 复测缓存右3位电芯条码50字（#2位）, 复测缓存右2位电芯条码50字（#2位）
@SET H51.03  ; 复测缓存右2位有料记忆（#2位）
@RSET H51.05  ; 复测缓存右3位有料记忆（#2位）
LD TR0
AND H51.06  ; 复测缓存左4位有料记忆（#1位）
@XFER(070) &50 E2_3300 E2_3200  ; 复测缓存左4位电芯条码50字（#1位）, 复测缓存左3位电芯条码50字（#1位）
@SET H51.04  ; 复测缓存左3位有料记忆（#1位）
@RSET H51.06  ; 复测缓存左4位有料记忆（#1位）
LD TR0
AND H51.07  ; 复测缓存右4位有料记忆（#2位）
@XFER(070) &50 E2_3350 E2_3250  ; 复测缓存右4位电芯条码50字（#2位）, 复测缓存右3位电芯条码50字（#2位）
@SET H51.05  ; 复测缓存右3位有料记忆（#2位）
@RSET H51.07  ; 复测缓存右4位有料记忆（#2位）

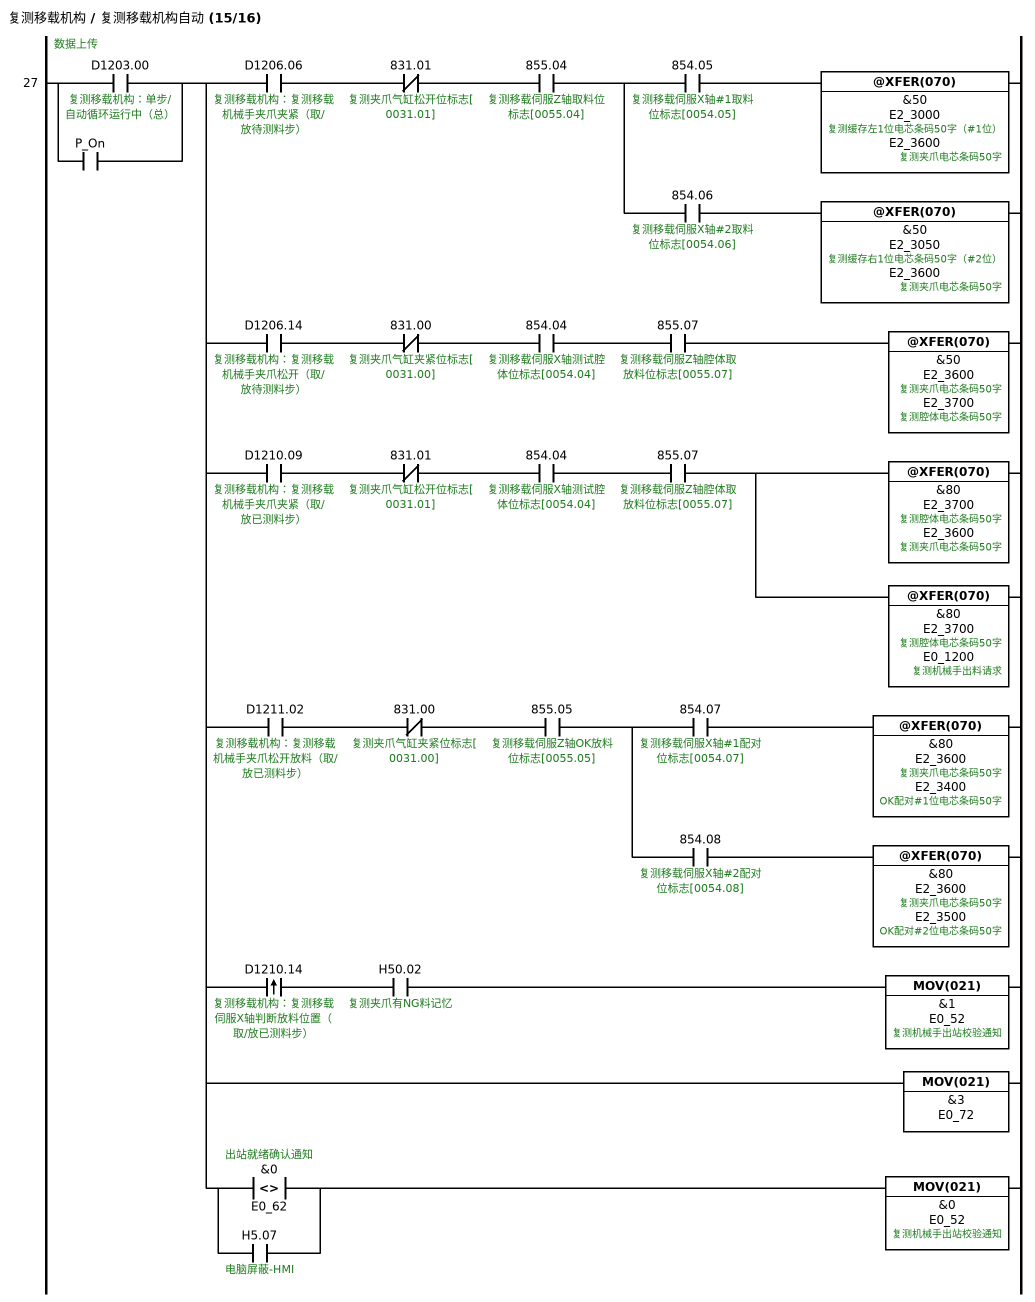
; rung 27: 数据上传
LD D1203.00  ; 复测移载机构：单步/自动循环运行中（总）
OR P_On
OUT TR0
AND D1206.06  ; 复测移载机构：复测移载机械手夹爪夹紧（取/放待测料步）
ANDNOT 831.01  ; 复测夹爪气缸松开位标志[0031.01]
AND 855.04  ; 复测移载伺服Z轴取料位标志[0055.04]
OUT TR1
AND 854.05  ; 复测移载伺服X轴#1取料位标志[0054.05]
@XFER(070) &50 E2_3000 E2_3600  ; 复测缓存左1位电芯条码50字（#1位）, 复测夹爪电芯条码50字
LD TR1
AND 854.06  ; 复测移载伺服X轴#2取料位标志[0054.06]
@XFER(070) &50 E2_3050 E2_3600  ; 复测缓存右1位电芯条码50字（#2位）, 复测夹爪电芯条码50字
LD TR0
AND D1206.14  ; 复测移载机构：复测移载机械手夹爪松开（取/放待测料步）
ANDNOT 831.00  ; 复测夹爪气缸夹紧位标志[0031.00]
AND 854.04  ; 复测移载伺服X轴测试腔体位标志[0054.04]
AND 855.07  ; 复测移载伺服Z轴腔体取放料位标志[0055.07]
@XFER(070) &50 E2_3600 E2_3700  ; 复测夹爪电芯条码50字, 复测腔体电芯条码50字
LD TR0
AND D1210.09  ; 复测移载机构：复测移载机械手夹爪夹紧（取/放已测料步）
ANDNOT 831.01  ; 复测夹爪气缸松开位标志[0031.01]
AND 854.04  ; 复测移载伺服X轴测试腔体位标志[0054.04]
AND 855.07  ; 复测移载伺服Z轴腔体取放料位标志[0055.07]
@XFER(070) &80 E2_3700 E2_3600  ; 复测腔体电芯条码50字, 复测夹爪电芯条码50字
@XFER(070) &80 E2_3700 E0_1200  ; 复测腔体电芯条码50字, 复测机械手出料请求
LD TR0
AND D1211.02  ; 复测移载机构：复测移载机械手夹爪松开放料（取/放已测料步）
ANDNOT 831.00  ; 复测夹爪气缸夹紧位标志[0031.00]
AND 855.05  ; 复测移载伺服Z轴OK放料位标志[0055.05]
OUT TR1
AND 854.07  ; 复测移载伺服X轴#1配对位标志[0054.07]
@XFER(070) &80 E2_3600 E2_3400  ; 复测夹爪电芯条码50字, OK配对#1位电芯条码50字
LD TR1
AND 854.08  ; 复测移载伺服X轴#2配对位标志[0054.08]
@XFER(070) &80 E2_3600 E2_3500  ; 复测夹爪电芯条码50字, OK配对#2位电芯条码50字
LD TR0
@AND D1210.14  ; 复测移载机构：复测移载伺服X轴判断放料位置（取/放已测料步）
AND H50.02  ; 复测夹爪有NG料记忆
MOV(021) &1 E0_52  ; 复测机械手出站校验通知
LD TR0
MOV(021) &3 E0_72
LD<>(305) &0 E0_62  ; 出站就绪确认通知
OR H5.07  ; 电脑屏蔽-HMI
ANDLD
MOV(021) &0 E0_52  ; 复测机械手出站校验通知

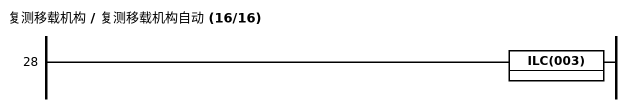
; rung 28
ILC(003)

### Section 复测移载机构手动

